LIN {X 0,Y 573.521,Z 268.884,A -85,B 0,C 180,E1 -2263.87,E2 -2263.87} C_VEL
LIN {X 0,Y 573.772,Z 242.194,A -85,B 0,C 180,E1 -2266.729,E2 -2266.729} C_VEL
LIN {X 0,Y 574.13,Z 213.422,A -85,B 0,C 180,E1 -2269.871,E2 -2269.871} C_VEL
LIN {X 0,Y 574.348,Z 185.649,A -85,B 0,C 180,E1 -2272.862,E2 -2272.862} C_VEL
LIN {X 0,Y 574.24,Z 177.963,A -85,B 0,C 180,E1 -2273.69,E2 -2273.69} C_VEL
LIN {X 0,Y 573.256,Z 173.17,A -85,B 0,C 180,E1 -2274.273,E2 -2274.273} C_VEL
LIN {X 0,Y 573.202,Z 173.086,A -85,B 0,C 180,E1 -2276.979,E2 -2276.979} C_VEL
LIN {X 0,Y 573.224,Z 173.084,A -85,B 0,C 180,E1 -2279.484,E2 -2279.484} C_VEL
LIN {X 0,Y 573.24,Z 173.075,A -85,B 0,C 180,E1 -2282.226,E2 -2282.226} C_VEL
LIN {X 0,Y 573.231,Z 173.08,A -85,B 0,C 180,E1 -2284.77,E2 -2284.77} C_VEL
LIN {X 0,Y 573.23,Z 173.077,A -85,B 0,C 180,E1 -2287.808,E2 -2287.808} C_VEL
LIN {X 0,Y 573.248,Z 173.076,A -85,B 0,C 180,E1 -2290.525,E2 -2290.525} C_VEL
LIN {X 0,Y 573.237,Z 173.076,A -85,B 0,C 180,E1 -2293.668,E2 -2293.668} C_VEL
LIN {X 0,Y 573.211,Z 173.083,A -85,B 0,C 180,E1 -2296.638,E2 -2296.638} C_VEL
LIN {X 0,Y 573.247,Z 173.075,A -85,B 0,C 180,E1 -2299.475,E2 -2299.475} C_VEL
LIN {X 0,Y 573.233,Z 173.076,A -85,B 0,C 180,E1 -2302.192,E2 -2302.192} C_VEL
LIN {X 0,Y 573.235,Z 173.079,A -85,B 0,C 180,E1 -2305.229,E2 -2305.229} C_VEL
LIN {X 0,Y 573.238,Z 173.076,A -85,B 0,C 180,E1 -2308.184,E2 -2308.184} C_VEL
LIN {X 0,Y 573.258,Z 173.081,A -85,B 0,C 180,E1 -2310.633,E2 -2310.633} C_VEL
LIN {X 0,Y 573.235,Z 173.075,A -85,B 0,C 180,E1 -2313.508,E2 -2313.508} C_VEL
LIN {X 0,Y 573.227,Z 173.079,A -85,B 0,C 180,E1 -2316.134,E2 -2316.134} C_VEL
LIN {X 0,Y 573.25,Z 173.075,A -85,B 0,C 180,E1 -2319.173,E2 -2319.173} C_VEL
LIN {X 0,Y 573.216,Z 173.078,A -85,B 0,C 180,E1 -2321.411,E2 -2321.411} C_VEL
LIN {X 0,Y 573.244,Z 173.074,A -85,B 0,C 180,E1 -2323.621,E2 -2323.621} C_VEL
LIN {X 0,Y 573.266,Z 173.073,A -85,B 0,C 180,E1 -2325.807,E2 -2325.807} C_VEL
LIN {X 0,Y 573.264,Z 173.077,A -85,B 0,C 180,E1 -2328.745,E2 -2328.745} C_VEL
LIN {X 0,Y 573.253,Z 173.073,A -85,B 0,C 180,E1 -2331.54,E2 -2331.54} C_VEL
LIN {X 0,Y 573.286,Z 173.078,A -85,B 0,C 180,E1 -2334.371,E2 -2334.371} C_VEL
LIN {X 0,Y 573.304,Z 173.072,A -85,B 0,C 180,E1 -2337.892,E2 -2337.892} C_VEL
LIN {X 0,Y 573.343,Z 173.26,A -85,B 0,C 180,E1 -2340.109,E2 -2340.109} C_VEL
LIN {X 0,Y 573.407,Z 187.13,A -85,B 0,C 180,E1 -2342.458,E2 -2342.458} C_VEL
LIN {X 0,Y 573.297,Z 202.339,A -85,B 0,C 180,E1 -2345.275,E2 -2345.275} C_VEL
LIN {X 0,Y 573.189,Z 217.748,A -85,B 0,C 180,E1 -2348.106,E2 -2348.106} C_VEL
LIN {X 0,Y 573.156,Z 223.495,A -85,B 0,C 180,E1 -2349.128,E2 -2349.128} C_VEL
LIN {X 0,Y 573.287,Z 224.818,A -85,B 0,C 180,E1 -2349.192,E2 -2349.192} C_VEL
LIN {X 0,Y 573.63,Z 230.578,A -85,B 0,C 180,E1 -2349.275,E2 -2349.275} C_VEL
LIN {X 0,Y 573.567,Z 299.116,A -85,B 0,C 180,E1 -2350.145,E2 -2350.145} C_VEL
LIN {X 0,Y 573.504,Z 308.495,A -85,B 0,C 180,E1 -2350.346,E2 -2350.346} C_VEL
LIN {X 0,Y 573.472,Z 317.469,A -85,B 0,C 180,E1 -2350.632,E2 -2350.632} C_VEL
LIN {X 0,Y 573.416,Z 327.573,A -85,B 0,C 180,E1 -2351.07,E2 -2351.07} C_VEL
LIN {X 0,Y 573.32,Z 337.992,A -85,B 0,C 180,E1 -2351.669,E2 -2351.669} C_VEL
LIN {X 0,Y 573.19,Z 347.471,A -85,B 0,C 180,E1 -2352.39,E2 -2352.39} C_VEL
LIN {X 0,Y 573.167,Z 353.388,A -85,B 0,C 180,E1 -2352.934,E2 -2352.934} C_VEL
LIN {X 0,Y 572.469,Z 357.587,A -85,B 0,C 180,E1 -2353.364,E2 -2353.364} C_VEL
LIN {X 0,Y 569.555,Z 363.708,A -85,B 0,C 180,E1 -2354.095,E2 -2354.095} C_VEL
LIN {X 0,Y 566.642,Z 369.015,A -85,B 0,C 180,E1 -2354.883,E2 -2354.883} C_VEL
LIN {X 0,Y 565.93,Z 371.801,A -85,B 0,C 180,E1 -2355.396,E2 -2355.396} C_VEL
LIN {X 0,Y 565.894,Z 376.999,A -85,B 0,C 180,E1 -2356.597,E2 -2356.597} C_VEL
LIN {X 0,Y 565.863,Z 379.373,A -85,B 0,C 180,E1 -2357.342,E2 -2357.342} C_VEL
LIN {X 0,Y 565.836,Z 381.091,A -85,B 0,C 180,E1 -2358.09,E2 -2358.09} C_VEL
LIN {X 0,Y 565.87,Z 382.685,A -85,B 0,C 180,E1 -2359.282,E2 -2359.282} C_VEL
LIN {X 0,Y 565.832,Z 382.89,A -85,B 0,C 180,E1 -2360.351,E2 -2360.351} C_VEL
LIN {X 0,Y 565.862,Z 382.12,A -85,B 0,C 180,E1 -2361.331,E2 -2361.331} C_VEL
LIN {X 0,Y 565.835,Z 381.35,A -85,B 0,C 180,E1 -2361.877,E2 -2361.877} C_VEL
LIN {X 0,Y 565.872,Z 379.63,A -85,B 0,C 180,E1 -2362.644,E2 -2362.644} C_VEL
LIN {X 0,Y 565.916,Z 375.822,A -85,B 0,C 180,E1 -2363.804,E2 -2363.804} C_VEL
LIN {X 0,Y 565.944,Z 371.347,A -85,B 0,C 180,E1 -2364.778,E2 -2364.778} C_VEL
LIN {X 0,Y 565.966,Z 366.81,A -85,B 0,C 180,E1 -2365.563,E2 -2365.563} C_VEL
LIN {X 0,Y 566.035,Z 361.227,A -85,B 0,C 180,E1 -2366.351,E2 -2366.351} C_VEL
LIN {X 0,Y 566.065,Z 356.174,A -85,B 0,C 180,E1 -2366.953,E2 -2366.953} C_VEL
LIN {X 0,Y 566.142,Z 349.213,A -85,B 0,C 180,E1 -2367.643,E2 -2367.643} C_VEL
LIN {X 0,Y 566.219,Z 342.41,A -85,B 0,C 180,E1 -2368.205,E2 -2368.205} C_VEL
LIN {X 0,Y 566.291,Z 334.823,A -85,B 0,C 180,E1 -2368.724,E2 -2368.724} C_VEL
LIN {X 0,Y 566.376,Z 326.258,A -85,B 0,C 180,E1 -2369.197,E2 -2369.197} C_VEL
LIN {X 0,Y 566.464,Z 316.793,A -85,B 0,C 180,E1 -2369.601,E2 -2369.601} C_VEL
LIN {X 0,Y 566.533,Z 307.068,A -85,B 0,C 180,E1 -2369.903,E2 -2369.903} C_VEL
LIN {X 0,Y 566.574,Z 295.422,A -85,B 0,C 180,E1 -2370.131,E2 -2370.131} C_VEL
LIN {X 0,Y 566.574,Z 227.134,A -85,B 0,C 180,E1 -2370.994,E2 -2370.994} C_VEL
LIN {X 0,Y 566.123,Z 223.733,A -85,B 0,C 180,E1 -2371.08,E2 -2371.08} C_VEL
LIN {X 0,Y 566.129,Z 219.328,A -85,B 0,C 180,E1 -2371.843,E2 -2371.843} C_VEL
LIN {X 0,Y 566.266,Z 203.344,A -85,B 0,C 180,E1 -2374.813,E2 -2374.813} C_VEL
LIN {X 0,Y 566.371,Z 187.85,A -85,B 0,C 180,E1 -2377.671,E2 -2377.671} C_VEL
LIN {X 0,Y 566.432,Z 175.809,A -85,B 0,C 180,E1 -2379.916,E2 -2379.916} C_VEL
LIN {X 0,Y 566.271,Z 173.97,A -85,B 0,C 180,E1 -2380.331,E2 -2380.331} C_VEL
LIN {X 0,Y 566.198,Z 173.953,A -85,B 0,C 180,E1 -2383.054,E2 -2383.054} C_VEL
LIN {X 0,Y 566.197,Z 173.958,A -85,B 0,C 180,E1 -2386.048,E2 -2386.048} C_VEL
LIN {X 0,Y 566.177,Z 173.954,A -85,B 0,C 180,E1 -2388.861,E2 -2388.861} C_VEL
LIN {X 0,Y 566.184,Z 173.962,A -85,B 0,C 180,E1 -2391.637,E2 -2391.637} C_VEL
LIN {X 0,Y 566.195,Z 173.953,A -85,B 0,C 180,E1 -2394.31,E2 -2394.31} C_VEL
LIN {X 0,Y 566.219,Z 173.949,A -85,B 0,C 180,E1 -2396.898,E2 -2396.898} C_VEL
LIN {X 0,Y 566.179,Z 173.961,A -85,B 0,C 180,E1 -2399.407,E2 -2399.407} C_VEL
LIN {X 0,Y 566.21,Z 173.954,A -85,B 0,C 180,E1 -2401.857,E2 -2401.857} C_VEL
LIN {X 0,Y 566.224,Z 173.948,A -85,B 0,C 180,E1 -2404.251,E2 -2404.251} C_VEL
LIN {X 0,Y 566.172,Z 173.955,A -85,B 0,C 180,E1 -2406.718,E2 -2406.718} C_VEL
LIN {X 0,Y 566.207,Z 173.956,A -85,B 0,C 180,E1 -2409.662,E2 -2409.662} C_VEL
LIN {X 0,Y 566.198,Z 173.952,A -85,B 0,C 180,E1 -2412.668,E2 -2412.668} C_VEL
LIN {X 0,Y 566.233,Z 173.952,A -85,B 0,C 180,E1 -2415.626,E2 -2415.626} C_VEL
LIN {X 0,Y 566.233,Z 173.949,A -85,B 0,C 180,E1 -2418.675,E2 -2418.675} C_VEL
LIN {X 0,Y 566.231,Z 173.953,A -85,B 0,C 180,E1 -2421.434,E2 -2421.434} C_VEL
LIN {X 0,Y 566.264,Z 173.943,A -85,B 0,C 180,E1 -2424.301,E2 -2424.301} C_VEL
LIN {X 0,Y 566.284,Z 173.941,A -85,B 0,C 180,E1 -2427.866,E2 -2427.866} C_VEL
LIN {X 0,Y 566.298,Z 173.943,A -85,B 0,C 180,E1 -2430.711,E2 -2430.711} C_VEL
LIN {X 0,Y 566.268,Z 173.949,A -85,B 0,C 180,E1 -2432.845,E2 -2432.845} C_VEL
LIN {X 0,Y 566.263,Z 173.944,A -85,B 0,C 180,E1 -2435.698,E2 -2435.698} C_VEL
LIN {X 0,Y 566.225,Z 173.952,A -85,B 0,C 180,E1 -2438.565,E2 -2438.565} C_VEL
LIN {X 0,Y 566.239,Z 173.948,A -85,B 0,C 180,E1 -2441.454,E2 -2441.454} C_VEL
LIN {X 0,Y 566.231,Z 173.951,A -85,B 0,C 180,E1 -2444.506,E2 -2444.506} C_VEL
LIN {X 0,Y 566.196,Z 173.954,A -85,B 0,C 180,E1 -2447.331,E2 -2447.331} C_VEL
LIN {X 0,Y 566.209,Z 173.953,A -85,B 0,C 180,E1 -2450.337,E2 -2450.337} C_VEL
LIN {X 0,Y 566.185,Z 173.954,A -85,B 0,C 180,E1 -2453.403,E2 -2453.403} C_VEL
LIN {X 0,Y 566.221,Z 173.948,A -85,B 0,C 180,E1 -2455.748,E2 -2455.748} C_VEL
LIN {X 0,Y 566.202,Z 173.954,A -85,B 0,C 180,E1 -2458.203,E2 -2458.203} C_VEL
LIN {X 0,Y 566.193,Z 173.955,A -85,B 0,C 180,E1 -2461.077,E2 -2461.077} C_VEL
LIN {X 0,Y 566.216,Z 173.951,A -85,B 0,C 180,E1 -2463.955,E2 -2463.955} C_VEL
LIN {X 0,Y 566.21,Z 173.959,A -85,B 0,C 180,E1 -2466.568,E2 -2466.568} C_VEL
LIN {X 0,Y 566.206,Z 173.951,A -85,B 0,C 180,E1 -2469.685,E2 -2469.685} C_VEL
LIN {X 0,Y 566.207,Z 173.955,A -85,B 0,C 180,E1 -2472.087,E2 -2472.087} C_VEL
LIN {X 0,Y 566.165,Z 173.956,A -85,B 0,C 180,E1 -2475.035,E2 -2475.035} C_VEL
LIN {X 0,Y 566.21,Z 173.956,A -85,B 0,C 180,E1 -2478.135,E2 -2478.135} C_VEL
LIN {X 0,Y 566.215,Z 173.952,A -85,B 0,C 180,E1 -2480.727,E2 -2480.727} C_VEL
LIN {X 0,Y 566.21,Z 173.953,A -85,B 0,C 180,E1 -2483.783,E2 -2483.783} C_VEL
LIN {X 0,Y 566.221,Z 173.957,A -85,B 0,C 180,E1 -2486.263,E2 -2486.263} C_VEL
LIN {X 0,Y 566.194,Z 173.952,A -85,B 0,C 180,E1 -2488.921,E2 -2488.921} C_VEL
LIN {X 0,Y 566.189,Z 173.952,A -85,B 0,C 180,E1 -2491.047,E2 -2491.047} C_VEL
LIN {X 0,Y 566.208,Z 173.951,A -85,B 0,C 180,E1 -2493.459,E2 -2493.459} C_VEL
LIN {X 0,Y 566.191,Z 173.958,A -85,B 0,C 180,E1 -2495.819,E2 -2495.819} C_VEL
LIN {X 0,Y 566.208,Z 173.95,A -85,B 0,C 180,E1 -2498.903,E2 -2498.903} C_VEL
LIN {X 0,Y 566.205,Z 173.951,A -85,B 0,C 180,E1 -2501.173,E2 -2501.173} C_VEL
LIN {X 0,Y 566.212,Z 173.952,A -85,B 0,C 180,E1 -2503.413,E2 -2503.413} C_VEL
LIN {X 0,Y 566.19,Z 173.955,A -85,B 0,C 180,E1 -2506.359,E2 -2506.359} C_VEL
LIN {X 0,Y 566.267,Z 173.943,A -85,B 0,C 180,E1 -2508.654,E2 -2508.654} C_VEL
LIN {X 0,Y 566.225,Z 173.952,A -85,B 0,C 180,E1 -2511.435,E2 -2511.435} C_VEL
LIN {X 0,Y 566.248,Z 173.947,A -85,B 0,C 180,E1 -2514.302,E2 -2514.302} C_VEL
LIN {X 0,Y 566.269,Z 173.95,A -85,B 0,C 180,E1 -2517.867,E2 -2517.867} C_VEL
LIN {X 0,Y 566.293,Z 173.939,A -85,B 0,C 180,E1 -2520.711,E2 -2520.711} C_VEL
LIN {X 0,Y 566.264,Z 173.943,A -85,B 0,C 180,E1 -2522.846,E2 -2522.846} C_VEL
LIN {X 0,Y 566.251,Z 173.953,A -85,B 0,C 180,E1 -2525.699,E2 -2525.699} C_VEL
LIN {X 0,Y 566.198,Z 173.951,A -85,B 0,C 180,E1 -2528.566,E2 -2528.566} C_VEL
LIN {X 0,Y 566.234,Z 173.956,A -85,B 0,C 180,E1 -2531.455,E2 -2531.455} C_VEL
LIN {X 0,Y 566.222,Z 173.948,A -85,B 0,C 180,E1 -2534.505,E2 -2534.505} C_VEL
LIN {X 0,Y 566.191,Z 173.961,A -85,B 0,C 180,E1 -2537.332,E2 -2537.332} C_VEL
LIN {X 0,Y 566.199,Z 173.951,A -85,B 0,C 180,E1 -2540.338,E2 -2540.338} C_VEL
LIN {X 0,Y 566.165,Z 173.965,A -85,B 0,C 180,E1 -2543.282,E2 -2543.282} C_VEL
LIN {X 0,Y 566.202,Z 173.954,A -85,B 0,C 180,E1 -2545.75,E2 -2545.75} C_VEL
LIN {X 0,Y 566.196,Z 173.951,A -85,B 0,C 180,E1 -2548.203,E2 -2548.203} C_VEL
LIN {X 0,Y 566.187,Z 173.961,A -85,B 0,C 180,E1 -2551.077,E2 -2551.077} C_VEL
LIN {X 0,Y 566.191,Z 173.954,A -85,B 0,C 180,E1 -2553.733,E2 -2553.733} C_VEL
LIN {X 0,Y 566.194,Z 173.954,A -85,B 0,C 180,E1 -2556.571,E2 -2556.571} C_VEL
LIN {X 0,Y 566.208,Z 173.951,A -85,B 0,C 180,E1 -2559.686,E2 -2559.686} C_VEL
LIN {X 0,Y 566.194,Z 173.96,A -85,B 0,C 180,E1 -2562.918,E2 -2562.918} C_VEL
LIN {X 0,Y 566.189,Z 173.952,A -85,B 0,C 180,E1 -2566.05,E2 -2566.05} C_VEL
LIN {X 0,Y 566.199,Z 173.956,A -85,B 0,C 180,E1 -2569.216,E2 -2569.216} C_VEL
LIN {X 0,Y 566.18,Z 173.954,A -85,B 0,C 180,E1 -2571.637,E2 -2571.637} C_VEL
LIN {X 0,Y 566.147,Z 173.96,A -85,B 0,C 180,E1 -2574.308,E2 -2574.308} C_VEL
LIN {X 0,Y 566.207,Z 173.959,A -85,B 0,C 180,E1 -2576.898,E2 -2576.898} C_VEL
LIN {X 0,Y 566.167,Z 173.958,A -85,B 0,C 180,E1 -2579.407,E2 -2579.407} C_VEL
LIN {X 0,Y 566.187,Z 173.955,A -85,B 0,C 180,E1 -2581.857,E2 -2581.857} C_VEL
LIN {X 0,Y 566.194,Z 173.959,A -85,B 0,C 180,E1 -2584.251,E2 -2584.251} C_VEL
LIN {X 0,Y 566.221,Z 174.083,A -85,B 0,C 180,E1 -2585.455,E2 -2585.455} C_VEL
LIN {X 0,Y 567.5,Z 179.942,A -85,B 0,C 180,E1 -2586.196,E2 -2586.196} C_VEL
LIN {X 0,Y 567.326,Z 199.749,A -85,B 0,C 180,E1 -2588.415,E2 -2588.415} C_VEL
LIN {X 0,Y 567.012,Z 225.162,A -85,B 0,C 180,E1 -2591.201,E2 -2591.201} C_VEL
LIN {X 0,Y 566.776,Z 248.942,A -85,B 0,C 180,E1 -2593.8,E2 -2593.8} C_VEL
LIN {X 0,Y 566.566,Z 268.903,A -85,B 0,C 180,E1 -2595.957,E2 -2595.957} C_VEL
LIN {X 0,Y 567.141,Z 274.771,A -85,B 0,C 180,E1 -2596.063,E2 -2596.063} C_VEL
LIN {X 0,Y 566.98,Z 378.978,A -85,B 0,C 180,E1 -2597.404,E2 -2597.404} C_VEL
LIN {X 0,Y 566.87,Z 392.239,A -85,B 0,C 180,E1 -2597.72,E2 -2597.72} C_VEL
LIN {X 0,Y 566.731,Z 405.171,A -85,B 0,C 180,E1 -2598.18,E2 -2598.18} C_VEL
LIN {X 0,Y 566.611,Z 417.257,A -85,B 0,C 180,E1 -2598.771,E2 -2598.771} C_VEL
LIN {X 0,Y 566.422,Z 429.493,A -85,B 0,C 180,E1 -2599.546,E2 -2599.546} C_VEL
LIN {X 0,Y 566.299,Z 439.653,A -85,B 0,C 180,E1 -2600.356,E2 -2600.356} C_VEL
LIN {X 0,Y 566.166,Z 448.791,A -85,B 0,C 180,E1 -2601.254,E2 -2601.254} C_VEL
LIN {X 0,Y 566.08,Z 457.693,A -85,B 0,C 180,E1 -2602.331,E2 -2602.331} C_VEL
LIN {X 0,Y 565.967,Z 464.959,A -85,B 0,C 180,E1 -2603.423,E2 -2603.423} C_VEL
LIN {X 0,Y 566.004,Z 469.682,A -85,B 0,C 180,E1 -2604.3,E2 -2604.3} C_VEL
LIN {X 0,Y 565.933,Z 474.375,A -85,B 0,C 180,E1 -2605.371,E2 -2605.371} C_VEL
LIN {X 0,Y 565.927,Z 477.959,A -85,B 0,C 180,E1 -2606.441,E2 -2606.441} C_VEL
LIN {X 0,Y 565.878,Z 479.809,A -85,B 0,C 180,E1 -2607.153,E2 -2607.153} C_VEL
LIN {X 0,Y 565.846,Z 482.185,A -85,B 0,C 180,E1 -2608.577,E2 -2608.577} C_VEL
LIN {X 0,Y 565.839,Z 483,A -85,B 0,C 180,E1 -2610,E2 -2610} C_VEL
LIN {X 0,Y 565.846,Z 482.185,A -85,B 0,C 180,E1 -2611.424,E2 -2611.424} C_VEL
LIN {X 0,Y 565.878,Z 479.809,A -85,B 0,C 180,E1 -2612.848,E2 -2612.848} C_VEL
LIN {X 0,Y 565.926,Z 476.894,A -85,B 0,C 180,E1 -2613.917,E2 -2613.917} C_VEL
LIN {X 0,Y 565.878,Z 472.947,A -85,B 0,C 180,E1 -2614.988,E2 -2614.988} C_VEL
LIN {X 0,Y 566.002,Z 467.865,A -85,B 0,C 180,E1 -2616.059,E2 -2616.059} C_VEL
LIN {X 0,Y 566.041,Z 461.465,A -85,B 0,C 180,E1 -2617.133,E2 -2617.133} C_VEL
LIN {X 0,Y 566.134,Z 453.474,A -85,B 0,C 180,E1 -2618.208,E2 -2618.208} C_VEL
LIN {X 0,Y 566.229,Z 445.33,A -85,B 0,C 180,E1 -2619.106,E2 -2619.106} C_VEL
LIN {X 0,Y 566.351,Z 435.394,A -85,B 0,C 180,E1 -2620.005,E2 -2620.005} C_VEL
LIN {X 0,Y 566.529,Z 424.285,A -85,B 0,C 180,E1 -2620.808,E2 -2620.808} C_VEL
LIN {X 0,Y 566.614,Z 413.166,A -85,B 0,C 180,E1 -2621.447,E2 -2621.447} C_VEL
LIN {X 0,Y 566.75,Z 400.97,A -85,B 0,C 180,E1 -2621.988,E2 -2621.988} C_VEL
LIN {X 0,Y 566.889,Z 388.159,A -85,B 0,C 180,E1 -2622.394,E2 -2622.394} C_VEL
LIN {X 0,Y 566.968,Z 374.575,A -85,B 0,C 180,E1 -2622.665,E2 -2622.665} C_VEL
LIN {X 0,Y 567.07,Z 272.9,A -85,B 0,C 180,E1 -2623.963,E2 -2623.963} C_VEL
LIN {X 0,Y 566.566,Z 268.885,A -85,B 0,C 180,E1 -2624.044,E2 -2624.044} C_VEL
LIN {X 0,Y 566.852,Z 241.138,A -85,B 0,C 180,E1 -2627.056,E2 -2627.056} C_VEL
LIN {X 0,Y 567.136,Z 214.637,A -85,B 0,C 180,E1 -2629.924,E2 -2629.924} C_VEL
LIN {X 0,Y 567.397,Z 186.667,A -85,B 0,C 180,E1 -2632.965,E2 -2632.965} C_VEL
LIN {X 0,Y 567.228,Z 178.993,A -85,B 0,C 180,E1 -2633.804,E2 -2633.804} C_VEL
LIN {X 0,Y 566.23,Z 174.085,A -85,B 0,C 180,E1 -2634.399,E2 -2634.399} C_VEL
LIN {X 0,Y 566.174,Z 173.964,A -85,B 0,C 180,E1 -2637.341,E2 -2637.341} C_VEL
LIN {X 0,Y 566.172,Z 173.959,A -85,B 0,C 180,E1 -2639.771,E2 -2639.771} C_VEL
LIN {X 0,Y 566.195,Z 173.953,A -85,B 0,C 180,E1 -2642.428,E2 -2642.428} C_VEL
LIN {X 0,Y 566.178,Z 173.962,A -85,B 0,C 180,E1 -2644.989,E2 -2644.989} C_VEL
LIN {X 0,Y 566.194,Z 173.957,A -85,B 0,C 180,E1 -2647.461,E2 -2647.461} C_VEL
LIN {X 0,Y 566.208,Z 173.951,A -85,B 0,C 180,E1 -2650.199,E2 -2650.199} C_VEL
LIN {X 0,Y 566.195,Z 173.962,A -85,B 0,C 180,E1 -2653.055,E2 -2653.055} C_VEL
LIN {X 0,Y 566.161,Z 173.956,A -85,B 0,C 180,E1 -2656.053,E2 -2656.053} C_VEL
LIN {X 0,Y 566.17,Z 173.964,A -85,B 0,C 180,E1 -2658.86,E2 -2658.86} C_VEL
LIN {X 0,Y 566.208,Z 173.952,A -85,B 0,C 180,E1 -2661.442,E2 -2661.442} C_VEL
LIN {X 0,Y 566.163,Z 173.958,A -85,B 0,C 180,E1 -2664.308,E2 -2664.308} C_VEL
LIN {X 0,Y 566.202,Z 173.96,A -85,B 0,C 180,E1 -2666.896,E2 -2666.896} C_VEL
LIN {X 0,Y 566.173,Z 173.956,A -85,B 0,C 180,E1 -2669.406,E2 -2669.406} C_VEL
LIN {X 0,Y 566.195,Z 173.952,A -85,B 0,C 180,E1 -2671.856,E2 -2671.856} C_VEL
LIN {X 0,Y 566.208,Z 173.954,A -85,B 0,C 180,E1 -2674.25,E2 -2674.25} C_VEL
LIN {X 0,Y 566.172,Z 173.963,A -85,B 0,C 180,E1 -2676.718,E2 -2676.718} C_VEL
LIN {X 0,Y 566.206,Z 173.951,A -85,B 0,C 180,E1 -2679.662,E2 -2679.662} C_VEL
LIN {X 0,Y 566.199,Z 173.96,A -85,B 0,C 180,E1 -2682.668,E2 -2682.668} C_VEL
LIN {X 0,Y 566.229,Z 173.948,A -85,B 0,C 180,E1 -2685.626,E2 -2685.626} C_VEL
LIN {X 0,Y 566.236,Z 173.953,A -85,B 0,C 180,E1 -2688.675,E2 -2688.675} C_VEL
LIN {X 0,Y 566.204,Z 173.951,A -85,B 0,C 180,E1 -2691.434,E2 -2691.434} C_VEL
LIN {X 0,Y 566.253,Z 173.954,A -85,B 0,C 180,E1 -2694.301,E2 -2694.301} C_VEL
LIN {X 0,Y 566.275,Z 173.947,A -85,B 0,C 180,E1 -2697.866,E2 -2697.866} C_VEL
LIN {X 0,Y 566.295,Z 174.105,A -85,B 0,C 180,E1 -2700.222,E2 -2700.222} C_VEL
LIN {X 0,Y 566.323,Z 185.594,A -85,B 0,C 180,E1 -2702.133,E2 -2702.133} C_VEL
LIN {X 0,Y 566.265,Z 199.749,A -85,B 0,C 180,E1 -2704.627,E2 -2704.627} C_VEL
LIN {X 0,Y 566.13,Z 215.239,A -85,B 0,C 180,E1 -2707.489,E2 -2707.489} C_VEL
LIN {X 0,Y 566.096,Z 223.554,A -85,B 0,C 180,E1 -2708.995,E2 -2708.995} C_VEL
LIN {X 0,Y 566.255,Z 225.049,A -85,B 0,C 180,E1 -2709.06,E2 -2709.06} C_VEL
LIN {X 0,Y 566.673,Z 230.673,A -85,B 0,C 180,E1 -2709.143,E2 -2709.143} C_VEL
LIN {X 0,Y 566.592,Z 299.184,A -85,B 0,C 180,E1 -2710.023,E2 -2710.023} C_VEL
LIN {X 0,Y 566.503,Z 308.568,A -85,B 0,C 180,E1 -2710.227,E2 -2710.227} C_VEL
LIN {X 0,Y 566.459,Z 318.268,A -85,B 0,C 180,E1 -2710.544,E2 -2710.544} C_VEL
LIN {X 0,Y 566.398,Z 328.843,A -85,B 0,C 180,E1 -2711.019,E2 -2711.019} C_VEL
LIN {X 0,Y 566.257,Z 338.974,A -85,B 0,C 180,E1 -2711.635,E2 -2711.635} C_VEL
LIN {X 0,Y 566.177,Z 347.221,A -85,B 0,C 180,E1 -2712.273,E2 -2712.273} C_VEL
LIN {X 0,Y 566.112,Z 354.026,A -85,B 0,C 180,E1 -2712.912,E2 -2712.912} C_VEL
LIN {X 0,Y 566.056,Z 360.479,A -85,B 0,C 180,E1 -2713.644,E2 -2713.644} C_VEL
LIN {X 0,Y 566.004,Z 366.081,A -85,B 0,C 180,E1 -2714.416,E2 -2714.416} C_VEL
LIN {X 0,Y 565.965,Z 370.295,A -85,B 0,C 180,E1 -2715.116,E2 -2715.116} C_VEL
LIN {X 0,Y 565.93,Z 371.801,A -85,B 0,C 180,E1 -2715.396,E2 -2715.396} C_VEL
LIN {X 0,Y 565.218,Z 374.462,A -85,B 0,C 180,E1 -2715.928,E2 -2715.928} C_VEL
LIN {X 0,Y 562.298,Z 378.055,A -85,B 0,C 180,E1 -2716.823,E2 -2716.823} C_VEL
LIN {X 0,Y 559.4,Z 380.595,A -85,B 0,C 180,E1 -2717.762,E2 -2717.762} C_VEL
LIN {X 0,Y 558.73,Z 381.603,A -85,B 0,C 180,E1 -2718.358,E2 -2718.358} C_VEL
LIN {X 0,Y 558.767,Z 382.733,A -85,B 0,C 180,E1 -2719.382,E2 -2719.382} C_VEL
LIN {X 0,Y 558.742,Z 382.772,A -85,B 0,C 180,E1 -2720.621,E2 -2720.621} C_VEL
LIN {X 0,Y 558.768,Z 381.983,A -85,B 0,C 180,E1 -2721.449,E2 -2721.449} C_VEL
LIN {X 0,Y 558.753,Z 380.771,A -85,B 0,C 180,E1 -2722.169,E2 -2722.169} C_VEL
LIN {X 0,Y 558.802,Z 377.599,A -85,B 0,C 180,E1 -2723.348,E2 -2723.348} C_VEL
LIN {X 0,Y 558.815,Z 374.671,A -85,B 0,C 180,E1 -2724.125,E2 -2724.125} C_VEL
LIN {X 0,Y 558.852,Z 371.446,A -85,B 0,C 180,E1 -2724.82,E2 -2724.82} C_VEL
LIN {X 0,Y 558.904,Z 366.312,A -85,B 0,C 180,E1 -2725.71,E2 -2725.71} C_VEL
LIN {X 0,Y 558.981,Z 360.62,A -85,B 0,C 180,E1 -2726.508,E2 -2726.508} C_VEL
LIN {X 0,Y 559.015,Z 355.499,A -85,B 0,C 180,E1 -2727.112,E2 -2727.112} C_VEL
LIN {X 0,Y 559.099,Z 348.338,A -85,B 0,C 180,E1 -2727.817,E2 -2727.817} C_VEL
LIN {X 0,Y 559.169,Z 341.423,A -85,B 0,C 180,E1 -2728.381,E2 -2728.381} C_VEL
LIN {X 0,Y 559.309,Z 333.196,A -85,B 0,C 180,E1 -2728.932,E2 -2728.932} C_VEL
LIN {X 0,Y 559.408,Z 323.85,A -85,B 0,C 180,E1 -2729.429,E2 -2729.429} C_VEL
LIN {X 0,Y 559.544,Z 312.135,A -85,B 0,C 180,E1 -2729.888,E2 -2729.888} C_VEL
LIN {X 0,Y 559.59,Z 301.336,A -85,B 0,C 180,E1 -2730.156,E2 -2730.156} C_VEL
LIN {X 0,Y 559.599,Z 274.915,A -85,B 0,C 180,E1 -2730.521,E2 -2730.521} C_VEL
LIN {X 0,Y 559.625,Z 227.896,A -85,B 0,C 180,E1 -2731.122,E2 -2731.122} C_VEL
LIN {X 0,Y 559.088,Z 223.909,A -85,B 0,C 180,E1 -2731.21,E2 -2731.21} C_VEL
LIN {X 0,Y 559.062,Z 221.829,A -85,B 0,C 180,E1 -2731.53,E2 -2731.53} C_VEL
LIN {X 0,Y 559.225,Z 206.44,A -85,B 0,C 180,E1 -2734.439,E2 -2734.439} C_VEL
LIN {X 0,Y 559.314,Z 190.38,A -85,B 0,C 180,E1 -2737.382,E2 -2737.382} C_VEL
LIN {X 0,Y 559.406,Z 176.654,A -85,B 0,C 180,E1 -2739.972,E2 -2739.972} C_VEL
LIN {X 0,Y 559.225,Z 174.852,A -85,B 0,C 180,E1 -2740.376,E2 -2740.376} C_VEL
LIN {X 0,Y 559.143,Z 174.833,A -85,B 0,C 180,E1 -2743.196,E2 -2743.196} C_VEL
LIN {X 0,Y 559.14,Z 174.834,A -85,B 0,C 180,E1 -2746.266,E2 -2746.266} C_VEL
LIN {X 0,Y 559.164,Z 174.828,A -85,B 0,C 180,E1 -2748.948,E2 -2748.948} C_VEL
LIN {X 0,Y 559.172,Z 174.829,A -85,B 0,C 180,E1 -2751.191,E2 -2751.191} C_VEL
LIN {X 0,Y 559.159,Z 174.835,A -85,B 0,C 180,E1 -2753.791,E2 -2753.791} C_VEL
LIN {X 0,Y 559.161,Z 174.828,A -85,B 0,C 180,E1 -2756.425,E2 -2756.425} C_VEL
LIN {X 0,Y 559.153,Z 174.831,A -85,B 0,C 180,E1 -2758.98,E2 -2758.98} C_VEL
LIN {X 0,Y 559.167,Z 174.836,A -85,B 0,C 180,E1 -2761.618,E2 -2761.618} C_VEL
LIN {X 0,Y 559.197,Z 174.827,A -85,B 0,C 180,E1 -2763.903,E2 -2763.903} C_VEL
LIN {X 0,Y 559.141,Z 174.83,A -85,B 0,C 180,E1 -2766.57,E2 -2766.57} C_VEL
LIN {X 0,Y 559.176,Z 174.836,A -85,B 0,C 180,E1 -2769.395,E2 -2769.395} C_VEL
LIN {X 0,Y 559.143,Z 174.835,A -85,B 0,C 180,E1 -2771.685,E2 -2771.685} C_VEL
LIN {X 0,Y 559.165,Z 174.829,A -85,B 0,C 180,E1 -2773.947,E2 -2773.947} C_VEL
LIN {X 0,Y 559.17,Z 174.827,A -85,B 0,C 180,E1 -2776.184,E2 -2776.184} C_VEL
LIN {X 0,Y 559.195,Z 174.832,A -85,B 0,C 180,E1 -2779.133,E2 -2779.133} C_VEL
LIN {X 0,Y 559.204,Z 174.823,A -85,B 0,C 180,E1 -2782.053,E2 -2782.053} C_VEL
LIN {X 0,Y 559.253,Z 174.823,A -85,B 0,C 180,E1 -2784.953,E2 -2784.953} C_VEL
LIN {X 0,Y 559.255,Z 174.817,A -85,B 0,C 180,E1 -2787.839,E2 -2787.839} C_VEL
LIN {X 0,Y 559.269,Z 174.819,A -85,B 0,C 180,E1 -2790.72,E2 -2790.72} C_VEL
LIN {X 0,Y 559.235,Z 174.826,A -85,B 0,C 180,E1 -2792.881,E2 -2792.881} C_VEL
LIN {X 0,Y 559.231,Z 174.82,A -85,B 0,C 180,E1 -2795.77,E2 -2795.77} C_VEL
LIN {X 0,Y 559.184,Z 174.83,A -85,B 0,C 180,E1 -2798.674,E2 -2798.674} C_VEL
LIN {X 0,Y 559.202,Z 174.824,A -85,B 0,C 180,E1 -2801.6,E2 -2801.6} C_VEL
LIN {X 0,Y 559.196,Z 174.829,A -85,B 0,C 180,E1 -2804.595,E2 -2804.595} C_VEL
LIN {X 0,Y 559.156,Z 174.829,A -85,B 0,C 180,E1 -2807.556,E2 -2807.556} C_VEL
LIN {X 0,Y 559.168,Z 174.827,A -85,B 0,C 180,E1 -2809.837,E2 -2809.837} C_VEL
LIN {X 0,Y 559.137,Z 174.833,A -85,B 0,C 180,E1 -2812.152,E2 -2812.152} C_VEL
LIN {X 0,Y 559.175,Z 174.829,A -85,B 0,C 180,E1 -2815.187,E2 -2815.187} C_VEL
LIN {X 0,Y 559.19,Z 174.824,A -85,B 0,C 180,E1 -2817.711,E2 -2817.711} C_VEL
LIN {X 0,Y 559.157,Z 174.832,A -85,B 0,C 180,E1 -2821.018,E2 -2821.018} C_VEL
LIN {X 0,Y 559.172,Z 174.828,A -85,B 0,C 180,E1 -2823.951,E2 -2823.951} C_VEL
LIN {X 0,Y 559.184,Z 174.834,A -85,B 0,C 180,E1 -2826.451,E2 -2826.451} C_VEL
LIN {X 0,Y 559.171,Z 174.83,A -85,B 0,C 180,E1 -2828.933,E2 -2828.933} C_VEL
LIN {X 0,Y 559.184,Z 174.826,A -85,B 0,C 180,E1 -2831.767,E2 -2831.767} C_VEL
LIN {X 0,Y 559.132,Z 174.836,A -85,B 0,C 180,E1 -2834.739,E2 -2834.739} C_VEL
LIN {X 0,Y 559.153,Z 174.829,A -85,B 0,C 180,E1 -2837.256,E2 -2837.256} C_VEL
LIN {X 0,Y 559.179,Z 174.833,A -85,B 0,C 180,E1 -2840.135,E2 -2840.135} C_VEL
LIN {X 0,Y 559.138,Z 174.832,A -85,B 0,C 180,E1 -2842.892,E2 -2842.892} C_VEL
LIN {X 0,Y 559.153,Z 174.83,A -85,B 0,C 180,E1 -2845.556,E2 -2845.556} C_VEL
LIN {X 0,Y 559.164,Z 174.837,A -85,B 0,C 180,E1 -2848.138,E2 -2848.138} C_VEL
LIN {X 0,Y 559.15,Z 174.832,A -85,B 0,C 180,E1 -2850.647,E2 -2850.647} C_VEL
LIN {X 0,Y 559.162,Z 174.828,A -85,B 0,C 180,E1 -2853.172,E2 -2853.172} C_VEL
LIN {X 0,Y 559.149,Z 174.831,A -85,B 0,C 180,E1 -2855.495,E2 -2855.495} C_VEL
LIN {X 0,Y 559.169,Z 174.828,A -85,B 0,C 180,E1 -2858.624,E2 -2858.624} C_VEL
LIN {X 0,Y 559.163,Z 174.827,A -85,B 0,C 180,E1 -2860.926,E2 -2860.926} C_VEL
LIN {X 0,Y 559.162,Z 174.838,A -85,B 0,C 180,E1 -2863.948,E2 -2863.948} C_VEL
LIN {X 0,Y 559.164,Z 174.833,A -85,B 0,C 180,E1 -2866.184,E2 -2866.184} C_VEL
LIN {X 0,Y 559.202,Z 174.824,A -85,B 0,C 180,E1 -2869.134,E2 -2869.134} C_VEL
LIN {X 0,Y 559.197,Z 174.829,A -85,B 0,C 180,E1 -2872.054,E2 -2872.054} C_VEL
LIN {X 0,Y 559.247,Z 174.818,A -85,B 0,C 180,E1 -2874.954,E2 -2874.954} C_VEL
LIN {X 0,Y 559.241,Z 174.826,A -85,B 0,C 180,E1 -2877.84,E2 -2877.84} C_VEL
LIN {X 0,Y 559.264,Z 174.815,A -85,B 0,C 180,E1 -2880.72,E2 -2880.72} C_VEL
LIN {X 0,Y 559.231,Z 174.82,A -85,B 0,C 180,E1 -2882.882,E2 -2882.882} C_VEL
LIN {X 0,Y 559.219,Z 174.827,A -85,B 0,C 180,E1 -2885.771,E2 -2885.771} C_VEL
LIN {X 0,Y 559.162,Z 174.828,A -85,B 0,C 180,E1 -2888.675,E2 -2888.675} C_VEL
LIN {X 0,Y 559.197,Z 174.831,A -85,B 0,C 180,E1 -2891.601,E2 -2891.601} C_VEL
LIN {X 0,Y 559.192,Z 174.824,A -85,B 0,C 180,E1 -2894.596,E2 -2894.596} C_VEL
LIN {X 0,Y 559.15,Z 174.836,A -85,B 0,C 180,E1 -2897.558,E2 -2897.558} C_VEL
LIN {X 0,Y 559.158,Z 174.831,A -85,B 0,C 180,E1 -2899.838,E2 -2899.838} C_VEL
LIN {X 0,Y 559.134,Z 174.831,A -85,B 0,C 180,E1 -2902.153,E2 -2902.153} C_VEL
LIN {X 0,Y 559.168,Z 174.837,A -85,B 0,C 180,E1 -2905.299,E2 -2905.299} C_VEL
LIN {X 0,Y 559.15,Z 174.832,A -85,B 0,C 180,E1 -2907.714,E2 -2907.714} C_VEL
LIN {X 0,Y 559.144,Z 174.83,A -85,B 0,C 180,E1 -2910.184,E2 -2910.184} C_VEL
LIN {X 0,Y 559.147,Z 174.833,A -85,B 0,C 180,E1 -2912.716,E2 -2912.716} C_VEL
LIN {X 0,Y 559.122,Z 174.839,A -85,B 0,C 180,E1 -2915.325,E2 -2915.325} C_VEL
LIN {X 0,Y 559.125,Z 174.832,A -85,B 0,C 180,E1 -2918.019,E2 -2918.019} C_VEL
LIN {X 0,Y 559.15,Z 174.835,A -85,B 0,C 180,E1 -2920.813,E2 -2920.813} C_VEL
LIN {X 0,Y 559.133,Z 174.832,A -85,B 0,C 180,E1 -2923.735,E2 -2923.735} C_VEL
LIN {X 0,Y 559.136,Z 174.839,A -85,B 0,C 180,E1 -2926.805,E2 -2926.805} C_VEL
LIN {X 0,Y 559.15,Z 174.834,A -85,B 0,C 180,E1 -2929.188,E2 -2929.188} C_VEL
LIN {X 0,Y 559.127,Z 174.832,A -85,B 0,C 180,E1 -2931.983,E2 -2931.983} C_VEL
LIN {X 0,Y 559.126,Z 174.842,A -85,B 0,C 180,E1 -2934.789,E2 -2934.789} C_VEL
LIN {X 0,Y 559.151,Z 174.832,A -85,B 0,C 180,E1 -2937.366,E2 -2937.366} C_VEL
LIN {X 0,Y 559.118,Z 174.837,A -85,B 0,C 180,E1 -2940.149,E2 -2940.149} C_VEL
LIN {X 0,Y 559.157,Z 174.836,A -85,B 0,C 180,E1 -2943.098,E2 -2943.098} C_VEL
LIN {X 0,Y 559.188,Z 175.008,A -85,B 0,C 180,E1 -2945.279,E2 -2945.279} C_VEL
LIN {X 0,Y 560.676,Z 182.426,A -85,B 0,C 180,E1 -2946.213,E2 -2946.213} C_VEL
LIN {X 0,Y 560.3,Z 207.599,A -85,B 0,C 180,E1 -2949.055,E2 -2949.055} C_VEL
LIN {X 0,Y 559.98,Z 231.628,A -85,B 0,C 180,E1 -2951.715,E2 -2951.715} C_VEL
LIN {X 0,Y 559.722,Z 255.6,A -85,B 0,C 180,E1 -2954.339,E2 -2954.339} C_VEL
LIN {X 0,Y 559.622,Z 268.904,A -85,B 0,C 180,E1 -2955.779,E2 -2955.779} C_VEL
LIN {X 0,Y 560.298,Z 276.56,A -85,B 0,C 180,E1 -2955.912,E2 -2955.912} C_VEL
LIN {X 0,Y 560.076,Z 378.978,A -85,B 0,C 180,E1 -2957.246,E2 -2957.246} C_VEL
LIN {X 0,Y 559.949,Z 392.238,A -85,B 0,C 180,E1 -2957.566,E2 -2957.566} C_VEL
LIN {X 0,Y 559.785,Z 405.172,A -85,B 0,C 180,E1 -2958.031,E2 -2958.031} C_VEL
LIN {X 0,Y 559.633,Z 417.856,A -85,B 0,C 180,E1 -2958.664,E2 -2958.664} C_VEL
LIN {X 0,Y 559.446,Z 429.495,A -85,B 0,C 180,E1 -2959.414,E2 -2959.414} C_VEL
LIN {X 0,Y 559.296,Z 439.653,A -85,B 0,C 180,E1 -2960.234,E2 -2960.234} C_VEL
LIN {X 0,Y 559.134,Z 448.791,A -85,B 0,C 180,E1 -2961.143,E2 -2961.143} C_VEL
LIN {X 0,Y 559.009,Z 457.692,A -85,B 0,C 180,E1 -2962.233,E2 -2962.233} C_VEL
LIN {X 0,Y 558.924,Z 463.743,A -85,B 0,C 180,E1 -2963.14,E2 -2963.14} C_VEL
LIN {X 0,Y 558.935,Z 469.682,A -85,B 0,C 180,E1 -2964.227,E2 -2964.227} C_VEL
LIN {X 0,Y 558.826,Z 474.375,A -85,B 0,C 180,E1 -2965.312,E2 -2965.312} C_VEL
LIN {X 0,Y 558.836,Z 477.96,A -85,B 0,C 180,E1 -2966.395,E2 -2966.395} C_VEL
LIN {X 0,Y 558.799,Z 479.808,A -85,B 0,C 180,E1 -2967.117,E2 -2967.117} C_VEL
LIN {X 0,Y 558.745,Z 482.184,A -85,B 0,C 180,E1 -2968.559,E2 -2968.559} C_VEL
LIN {X 0,Y 558.74,Z 483,A -85,B 0,C 180,E1 -2970.001,E2 -2970.001} C_VEL
LIN {X 0,Y 558.745,Z 482.184,A -85,B 0,C 180,E1 -2971.442,E2 -2971.442} C_VEL
LIN {X 0,Y 558.799,Z 479.809,A -85,B 0,C 180,E1 -2972.884,E2 -2972.884} C_VEL
LIN {X 0,Y 558.844,Z 476.894,A -85,B 0,C 180,E1 -2973.967,E2 -2973.967} C_VEL
LIN {X 0,Y 558.798,Z 472.946,A -85,B 0,C 180,E1 -2975.051,E2 -2975.051} C_VEL
LIN {X 0,Y 558.921,Z 467.865,A -85,B 0,C 180,E1 -2976.136,E2 -2976.136} C_VEL
LIN {X 0,Y 558.978,Z 461.464,A -85,B 0,C 180,E1 -2977.223,E2 -2977.223} C_VEL
LIN {X 0,Y 559.099,Z 453.474,A -85,B 0,C 180,E1 -2978.312,E2 -2978.312} C_VEL
LIN {X 0,Y 559.195,Z 445.33,A -85,B 0,C 180,E1 -2979.221,E2 -2979.221} C_VEL
LIN {X 0,Y 559.362,Z 435.393,A -85,B 0,C 180,E1 -2980.131,E2 -2980.131} C_VEL
LIN {X 0,Y 559.538,Z 424.391,A -85,B 0,C 180,E1 -2980.937,E2 -2980.937} C_VEL
LIN {X 0,Y 559.673,Z 412.45,A -85,B 0,C 180,E1 -2981.628,E2 -2981.628} C_VEL
LIN {X 0,Y 559.825,Z 399.757,A -85,B 0,C 180,E1 -2982.185,E2 -2982.185} C_VEL
LIN {X 0,Y 559.987,Z 386.329,A -85,B 0,C 180,E1 -2982.596,E2 -2982.596} C_VEL
LIN {X 0,Y 560.066,Z 373.057,A -85,B 0,C 180,E1 -2982.847,E2 -2982.847} C_VEL
LIN {X 0,Y 560.196,Z 273.574,A -85,B 0,C 180,E1 -2984.129,E2 -2984.129} C_VEL
LIN {X 0,Y 559.603,Z 268.886,A -85,B 0,C 180,E1 -2984.223,E2 -2984.223} C_VEL
LIN {X 0,Y 559.886,Z 240.146,A -85,B 0,C 180,E1 -2987.33,E2 -2987.33} C_VEL
LIN {X 0,Y 560.175,Z 212.24,A -85,B 0,C 180,E1 -2990.375,E2 -2990.375} C_VEL
LIN {X 0,Y 560.466,Z 185.891,A -85,B 0,C 180,E1 -2993.266,E2 -2993.266} C_VEL
LIN {X 0,Y 560.344,Z 180.71,A -85,B 0,C 180,E1 -2993.84,E2 -2993.84} C_VEL
LIN {X 0,Y 559.167,Z 174.943,A -85,B 0,C 180,E1 -2994.553,E2 -2994.553} C_VEL
LIN {X 0,Y 559.138,Z 174.838,A -85,B 0,C 180,E1 -2996.904,E2 -2996.904} C_VEL
LIN {X 0,Y 559.122,Z 174.836,A -85,B 0,C 180,E1 -2999.852,E2 -2999.852} C_VEL
LIN {X 0,Y 559.15,Z 174.833,A -85,B 0,C 180,E1 -3002.716,E2 -3002.716} C_VEL
LIN {X 0,Y 559.124,Z 174.841,A -85,B 0,C 180,E1 -3005.325,E2 -3005.325} C_VEL
LIN {X 0,Y 559.13,Z 174.833,A -85,B 0,C 180,E1 -3008.018,E2 -3008.018} C_VEL
LIN {X 0,Y 559.156,Z 174.835,A -85,B 0,C 180,E1 -3010.813,E2 -3010.813} C_VEL
LIN {X 0,Y 559.138,Z 174.832,A -85,B 0,C 180,E1 -3013.734,E2 -3013.734} C_VEL
LIN {X 0,Y 559.133,Z 174.839,A -85,B 0,C 180,E1 -3016.805,E2 -3016.805} C_VEL
LIN {X 0,Y 559.156,Z 174.834,A -85,B 0,C 180,E1 -3019.187,E2 -3019.187} C_VEL
LIN {X 0,Y 559.131,Z 174.832,A -85,B 0,C 180,E1 -3021.982,E2 -3021.982} C_VEL
LIN {X 0,Y 559.133,Z 174.84,A -85,B 0,C 180,E1 -3024.787,E2 -3024.787} C_VEL
LIN {X 0,Y 559.154,Z 174.831,A -85,B 0,C 180,E1 -3027.365,E2 -3027.365} C_VEL
LIN {X 0,Y 559.144,Z 174.832,A -85,B 0,C 180,E1 -3030.144,E2 -3030.144} C_VEL
LIN {X 0,Y 559.167,Z 174.83,A -85,B 0,C 180,E1 -3033.173,E2 -3033.173} C_VEL
LIN {X 0,Y 559.156,Z 174.829,A -85,B 0,C 180,E1 -3035.495,E2 -3035.495} C_VEL
LIN {X 0,Y 559.173,Z 174.836,A -85,B 0,C 180,E1 -3038.624,E2 -3038.624} C_VEL
LIN {X 0,Y 559.161,Z 174.833,A -85,B 0,C 180,E1 -3040.926,E2 -3040.926} C_VEL
LIN {X 0,Y 559.162,Z 174.831,A -85,B 0,C 180,E1 -3043.947,E2 -3043.947} C_VEL
LIN {X 0,Y 559.166,Z 174.834,A -85,B 0,C 180,E1 -3046.184,E2 -3046.184} C_VEL
LIN {X 0,Y 559.194,Z 174.826,A -85,B 0,C 180,E1 -3049.133,E2 -3049.133} C_VEL
LIN {X 0,Y 559.195,Z 174.83,A -85,B 0,C 180,E1 -3052.053,E2 -3052.053} C_VEL
LIN {X 0,Y 559.247,Z 174.82,A -85,B 0,C 180,E1 -3054.953,E2 -3054.953} C_VEL
LIN {X 0,Y 559.247,Z 174.823,A -85,B 0,C 180,E1 -3057.839,E2 -3057.839} C_VEL
LIN {X 0,Y 559.243,Z 175.009,A -85,B 0,C 180,E1 -3060.315,E2 -3060.315} C_VEL
LIN {X 0,Y 559.246,Z 185.03,A -85,B 0,C 180,E1 -3061.98,E2 -3061.98} C_VEL
LIN {X 0,Y 559.191,Z 194.423,A -85,B 0,C 180,E1 -3063.603,E2 -3063.603} C_VEL
LIN {X 0,Y 559.19,Z 206.905,A -85,B 0,C 180,E1 -3065.77,E2 -3065.77} C_VEL
LIN {X 0,Y 559.073,Z 220.513,A -85,B 0,C 180,E1 -3068.312,E2 -3068.312} C_VEL
LIN {X 0,Y 559.051,Z 223.643,A -85,B 0,C 180,E1 -3068.858,E2 -3068.858} C_VEL
LIN {X 0,Y 559.391,Z 226.368,A -85,B 0,C 180,E1 -3068.944,E2 -3068.944} C_VEL
LIN {X 0,Y 559.713,Z 232.565,A -85,B 0,C 180,E1 -3069.03,E2 -3069.03} C_VEL
LIN {X 0,Y 559.611,Z 299.27,A -85,B 0,C 180,E1 -3069.898,E2 -3069.898} C_VEL
LIN {X 0,Y 559.55,Z 307.747,A -85,B 0,C 180,E1 -3070.082,E2 -3070.082} C_VEL
LIN {X 0,Y 559.487,Z 316.472,A -85,B 0,C 180,E1 -3070.357,E2 -3070.357} C_VEL
LIN {X 0,Y 559.393,Z 324.222,A -85,B 0,C 180,E1 -3070.679,E2 -3070.679} C_VEL
LIN {X 0,Y 559.284,Z 332.431,A -85,B 0,C 180,E1 -3071.112,E2 -3071.112} C_VEL
LIN {X 0,Y 559.221,Z 339.933,A -85,B 0,C 180,E1 -3071.6,E2 -3071.6} C_VEL
LIN {X 0,Y 559.104,Z 348.031,A -85,B 0,C 180,E1 -3072.246,E2 -3072.246} C_VEL
LIN {X 0,Y 559.048,Z 354.698,A -85,B 0,C 180,E1 -3072.893,E2 -3072.893} C_VEL
LIN {X 0,Y 558.973,Z 361.044,A -85,B 0,C 180,E1 -3073.635,E2 -3073.635} C_VEL
LIN {X 0,Y 558.903,Z 366.947,A -85,B 0,C 180,E1 -3074.478,E2 -3074.478} C_VEL
LIN {X 0,Y 558.856,Z 371.992,A -85,B 0,C 180,E1 -3075.379,E2 -3075.379} C_VEL
LIN {X 0,Y 558.818,Z 376.612,A -85,B 0,C 180,E1 -3076.437,E2 -3076.437} C_VEL
LIN {X 0,Y 558.764,Z 379.981,A -85,B 0,C 180,E1 -3077.569,E2 -3077.569} C_VEL
LIN {X 0,Y 558.73,Z 381.603,A -85,B 0,C 180,E1 -3078.358,E2 -3078.358} C_VEL
LIN {X 0,Y 558.057,Z 382.406,A -85,B 0,C 180,E1 -3078.955,E2 -3078.955} C_VEL
LIN {X 0,Y 556.457,Z 382.878,A -85,B 0,C 180,E1 -3079.542,E2 -3079.542} C_VEL
LIN {X 0,Y 552.741,Z 382.733,A -85,B 0,C 180,E1 -3080.715,E2 -3080.715} C_VEL
LIN {X 0,Y 551.732,Z 382.18,A -85,B 0,C 180,E1 -3081.319,E2 -3081.319} C_VEL
LIN {X 0,Y 551.667,Z 381.902,A -85,B 0,C 180,E1 -3081.523,E2 -3081.523} C_VEL
LIN {X 0,Y 551.693,Z 379.249,A -85,B 0,C 180,E1 -3082.863,E2 -3082.863} C_VEL
LIN {X 0,Y 551.739,Z 376.483,A -85,B 0,C 180,E1 -3083.735,E2 -3083.735} C_VEL
LIN {X 0,Y 551.783,Z 371.601,A -85,B 0,C 180,E1 -3084.854,E2 -3084.854} C_VEL
LIN {X 0,Y 551.841,Z 365.885,A -85,B 0,C 180,E1 -3085.861,E2 -3085.861} C_VEL
LIN {X 0,Y 551.924,Z 359.816,A -85,B 0,C 180,E1 -3086.712,E2 -3086.712} C_VEL
LIN {X 0,Y 552.031,Z 351.008,A -85,B 0,C 180,E1 -3087.69,E2 -3087.69} C_VEL
LIN {X 0,Y 552.168,Z 342.828,A -85,B 0,C 180,E1 -3088.398,E2 -3088.398} C_VEL
LIN {X 0,Y 552.304,Z 333.849,A -85,B 0,C 180,E1 -3089.021,E2 -3089.021} C_VEL
LIN {X 0,Y 552.419,Z 324.397,A -85,B 0,C 180,E1 -3089.537,E2 -3089.537} C_VEL
LIN {X 0,Y 552.554,Z 313.01,A -85,B 0,C 180,E1 -3089.997,E2 -3089.997} C_VEL
LIN {X 0,Y 552.62,Z 301.864,A -85,B 0,C 180,E1 -3090.284,E2 -3090.284} C_VEL
LIN {X 0,Y 552.662,Z 272.587,A -85,B 0,C 180,E1 -3090.694,E2 -3090.694} C_VEL
LIN {X 0,Y 552.664,Z 228.414,A -85,B 0,C 180,E1 -3091.27,E2 -3091.27} C_VEL
LIN {X 0,Y 552.059,Z 223.902,A -85,B 0,C 180,E1 -3091.383,E2 -3091.383} C_VEL
LIN {X 0,Y 552.052,Z 217.199,A -85,B 0,C 180,E1 -3092.584,E2 -3092.584} C_VEL
LIN {X 0,Y 552.229,Z 203.398,A -85,B 0,C 180,E1 -3095.199,E2 -3095.199} C_VEL
LIN {X 0,Y 552.318,Z 188.67,A -85,B 0,C 180,E1 -3097.915,E2 -3097.915} C_VEL
LIN {X 0,Y 552.414,Z 178.391,A -85,B 0,C 180,E1 -3099.858,E2 -3099.858} C_VEL
LIN {X 0,Y 552.192,Z 175.76,A -85,B 0,C 180,E1 -3100.411,E2 -3100.411} C_VEL
LIN {X 0,Y 552.09,Z 175.714,A -85,B 0,C 180,E1 -3103.481,E2 -3103.481} C_VEL
LIN {X 0,Y 552.105,Z 175.708,A -85,B 0,C 180,E1 -3106.576,E2 -3106.576} C_VEL
LIN {X 0,Y 552.108,Z 175.713,A -85,B 0,C 180,E1 -3109.519,E2 -3109.519} C_VEL
LIN {X 0,Y 552.091,Z 175.71,A -85,B 0,C 180,E1 -3112.336,E2 -3112.336} C_VEL
LIN {X 0,Y 552.118,Z 175.707,A -85,B 0,C 180,E1 -3115.053,E2 -3115.053} C_VEL
LIN {X 0,Y 552.115,Z 175.714,A -85,B 0,C 180,E1 -3117.681,E2 -3117.681} C_VEL
LIN {X 0,Y 552.11,Z 175.707,A -85,B 0,C 180,E1 -3120.235,E2 -3120.235} C_VEL
LIN {X 0,Y 552.144,Z 175.704,A -85,B 0,C 180,E1 -3122.998,E2 -3122.998} C_VEL
LIN {X 0,Y 552.113,Z 175.711,A -85,B 0,C 180,E1 -3125.161,E2 -3125.161} C_VEL
LIN {X 0,Y 552.124,Z 175.704,A -85,B 0,C 180,E1 -3128.337,E2 -3128.337} C_VEL
LIN {X 0,Y 552.15,Z 175.702,A -85,B 0,C 180,E1 -3130.674,E2 -3130.674} C_VEL
LIN {X 0,Y 552.115,Z 175.709,A -85,B 0,C 180,E1 -3133.737,E2 -3133.737} C_VEL
LIN {X 0,Y 552.134,Z 175.704,A -85,B 0,C 180,E1 -3136.004,E2 -3136.004} C_VEL
LIN {X 0,Y 552.162,Z 175.705,A -85,B 0,C 180,E1 -3138.993,E2 -3138.993} C_VEL
LIN {X 0,Y 552.158,Z 175.701,A -85,B 0,C 180,E1 -3141.951,E2 -3141.951} C_VEL
LIN {X 0,Y 552.228,Z 175.697,A -85,B 0,C 180,E1 -3144.888,E2 -3144.888} C_VEL
LIN {X 0,Y 552.226,Z 175.693,A -85,B 0,C 180,E1 -3147.811,E2 -3147.811} C_VEL
LIN {X 0,Y 552.239,Z 175.694,A -85,B 0,C 180,E1 -3150.729,E2 -3150.729} C_VEL
LIN {X 0,Y 552.202,Z 175.703,A -85,B 0,C 180,E1 -3152.918,E2 -3152.918} C_VEL
LIN {X 0,Y 552.2,Z 175.695,A -85,B 0,C 180,E1 -3155.843,E2 -3155.843} C_VEL
LIN {X 0,Y 552.155,Z 175.708,A -85,B 0,C 180,E1 -3158.785,E2 -3158.785} C_VEL
LIN {X 0,Y 552.159,Z 175.7,A -85,B 0,C 180,E1 -3161.75,E2 -3161.75} C_VEL
LIN {X 0,Y 552.133,Z 175.711,A -85,B 0,C 180,E1 -3164.748,E2 -3164.748} C_VEL
LIN {X 0,Y 552.107,Z 175.707,A -85,B 0,C 180,E1 -3167.788,E2 -3167.788} C_VEL
LIN {X 0,Y 552.127,Z 175.705,A -85,B 0,C 180,E1 -3170.101,E2 -3170.101} C_VEL
LIN {X 0,Y 552.092,Z 175.714,A -85,B 0,C 180,E1 -3172.45,E2 -3172.45} C_VEL
LIN {X 0,Y 552.152,Z 175.702,A -85,B 0,C 180,E1 -3175.35,E2 -3175.35} C_VEL
LIN {X 0,Y 552.122,Z 175.707,A -85,B 0,C 180,E1 -3178.097,E2 -3178.097} C_VEL
LIN {X 0,Y 552.102,Z 175.717,A -85,B 0,C 180,E1 -3180.608,E2 -3180.608} C_VEL
LIN {X 0,Y 552.123,Z 175.706,A -85,B 0,C 180,E1 -3183.184,E2 -3183.184} C_VEL
LIN {X 0,Y 552.107,Z 175.708,A -85,B 0,C 180,E1 -3185.841,E2 -3185.841} C_VEL
LIN {X 0,Y 552.118,Z 175.707,A -85,B 0,C 180,E1 -3189.061,E2 -3189.061} C_VEL
LIN {X 0,Y 552.133,Z 175.703,A -85,B 0,C 180,E1 -3191.444,E2 -3191.444} C_VEL
LIN {X 0,Y 552.089,Z 175.716,A -85,B 0,C 180,E1 -3194.532,E2 -3194.532} C_VEL
LIN {X 0,Y 552.123,Z 175.705,A -85,B 0,C 180,E1 -3197.584,E2 -3197.584} C_VEL
LIN {X 0,Y 552.127,Z 175.711,A -85,B 0,C 180,E1 -3200.473,E2 -3200.473} C_VEL
LIN {X 0,Y 552.106,Z 175.707,A -85,B 0,C 180,E1 -3203.315,E2 -3203.315} C_VEL
LIN {X 0,Y 552.132,Z 175.709,A -85,B 0,C 180,E1 -3205.94,E2 -3205.94} C_VEL
LIN {X 0,Y 552.11,Z 175.71,A -85,B 0,C 180,E1 -3208.54,E2 -3208.54} C_VEL
LIN {X 0,Y 552.118,Z 175.706,A -85,B 0,C 180,E1 -3211.437,E2 -3211.437} C_VEL
LIN {X 0,Y 552.121,Z 175.71,A -85,B 0,C 180,E1 -3214.356,E2 -3214.356} C_VEL
LIN {X 0,Y 552.102,Z 175.708,A -85,B 0,C 180,E1 -3216.758,E2 -3216.758} C_VEL
LIN {X 0,Y 552.118,Z 175.705,A -85,B 0,C 180,E1 -3219.12,E2 -3219.12} C_VEL
LIN {X 0,Y 552.123,Z 175.707,A -85,B 0,C 180,E1 -3221.445,E2 -3221.445} C_VEL
LIN {X 0,Y 552.111,Z 175.713,A -85,B 0,C 180,E1 -3223.738,E2 -3223.738} C_VEL
LIN {X 0,Y 552.127,Z 175.712,A -85,B 0,C 180,E1 -3226.005,E2 -3226.005} C_VEL
LIN {X 0,Y 552.17,Z 175.699,A -85,B 0,C 180,E1 -3228.994,E2 -3228.994} C_VEL
LIN {X 0,Y 552.151,Z 175.708,A -85,B 0,C 180,E1 -3231.952,E2 -3231.952} C_VEL
LIN {X 0,Y 552.221,Z 175.693,A -85,B 0,C 180,E1 -3234.889,E2 -3234.889} C_VEL
LIN {X 0,Y 552.213,Z 175.702,A -85,B 0,C 180,E1 -3237.812,E2 -3237.812} C_VEL
LIN {X 0,Y 552.234,Z 175.691,A -85,B 0,C 180,E1 -3240.73,E2 -3240.73} C_VEL
LIN {X 0,Y 552.198,Z 175.696,A -85,B 0,C 180,E1 -3242.918,E2 -3242.918} C_VEL
LIN {X 0,Y 552.189,Z 175.702,A -85,B 0,C 180,E1 -3245.844,E2 -3245.844} C_VEL
LIN {X 0,Y 552.137,Z 175.703,A -85,B 0,C 180,E1 -3248.786,E2 -3248.786} C_VEL
LIN {X 0,Y 552.155,Z 175.706,A -85,B 0,C 180,E1 -3251.751,E2 -3251.751} C_VEL
LIN {X 0,Y 552.128,Z 175.705,A -85,B 0,C 180,E1 -3254.749,E2 -3254.749} C_VEL
LIN {X 0,Y 552.1,Z 175.711,A -85,B 0,C 180,E1 -3257.789,E2 -3257.789} C_VEL
LIN {X 0,Y 552.119,Z 175.706,A -85,B 0,C 180,E1 -3260.102,E2 -3260.102} C_VEL
LIN {X 0,Y 552.085,Z 175.709,A -85,B 0,C 180,E1 -3262.452,E2 -3262.452} C_VEL
LIN {X 0,Y 552.148,Z 175.71,A -85,B 0,C 180,E1 -3265.351,E2 -3265.351} C_VEL
LIN {X 0,Y 552.09,Z 175.709,A -85,B 0,C 180,E1 -3268.1,E2 -3268.1} C_VEL
LIN {X 0,Y 552.096,Z 175.71,A -85,B 0,C 180,E1 -3270.61,E2 -3270.61} C_VEL
LIN {X 0,Y 552.101,Z 175.717,A -85,B 0,C 180,E1 -3273.187,E2 -3273.187} C_VEL
LIN {X 0,Y 552.08,Z 175.711,A -85,B 0,C 180,E1 -3275.844,E2 -3275.844} C_VEL
LIN {X 0,Y 552.115,Z 175.716,A -85,B 0,C 180,E1 -3279.062,E2 -3279.062} C_VEL
LIN {X 0,Y 552.115,Z 175.709,A -85,B 0,C 180,E1 -3281.447,E2 -3281.447} C_VEL
LIN {X 0,Y 552.087,Z 175.712,A -85,B 0,C 180,E1 -3284.532,E2 -3284.532} C_VEL
LIN {X 0,Y 552.104,Z 175.708,A -85,B 0,C 180,E1 -3287.588,E2 -3287.588} C_VEL
LIN {X 0,Y 552.127,Z 175.707,A -85,B 0,C 180,E1 -3290.474,E2 -3290.474} C_VEL
LIN {X 0,Y 552.096,Z 175.711,A -85,B 0,C 180,E1 -3293.319,E2 -3293.319} C_VEL
LIN {X 0,Y 552.122,Z 175.706,A -85,B 0,C 180,E1 -3295.94,E2 -3295.94} C_VEL
LIN {X 0,Y 552.118,Z 175.713,A -85,B 0,C 180,E1 -3298.542,E2 -3298.542} C_VEL
LIN {X 0,Y 552.101,Z 175.71,A -85,B 0,C 180,E1 -3301.443,E2 -3301.443} C_VEL
LIN {X 0,Y 552.104,Z 175.712,A -85,B 0,C 180,E1 -3303.543,E2 -3303.543} C_VEL
LIN {X 0,Y 552.155,Z 175.894,A -85,B 0,C 180,E1 -3305.089,E2 -3305.089} C_VEL
LIN {X 0,Y 553.826,Z 184.429,A -85,B 0,C 180,E1 -3306.175,E2 -3306.175} C_VEL
LIN {X 0,Y 553.381,Z 210.669,A -85,B 0,C 180,E1 -3309.17,E2 -3309.17} C_VEL
LIN {X 0,Y 552.943,Z 238.071,A -85,B 0,C 180,E1 -3312.24,E2 -3312.24} C_VEL
LIN {X 0,Y 552.609,Z 265.421,A -85,B 0,C 180,E1 -3315.265,E2 -3315.265} C_VEL
LIN {X 0,Y 552.622,Z 268.875,A -85,B 0,C 180,E1 -3315.618,E2 -3315.618} C_VEL
LIN {X 0,Y 553.391,Z 277.159,A -85,B 0,C 180,E1 -3315.756,E2 -3315.756} C_VEL
LIN {X 0,Y 553.139,Z 378.697,A -85,B 0,C 180,E1 -3317.084,E2 -3317.084} C_VEL
LIN {X 0,Y 553.03,Z 392.137,A -85,B 0,C 180,E1 -3317.408,E2 -3317.408} C_VEL
LIN {X 0,Y 552.812,Z 404.37,A -85,B 0,C 180,E1 -3317.845,E2 -3317.845} C_VEL
LIN {X 0,Y 552.689,Z 416.677,A -85,B 0,C 180,E1 -3318.45,E2 -3318.45} C_VEL
LIN {X 0,Y 552.49,Z 428.201,A -85,B 0,C 180,E1 -3319.186,E2 -3319.186} C_VEL
LIN {X 0,Y 552.276,Z 438.612,A -85,B 0,C 180,E1 -3320.016,E2 -3320.016} C_VEL
LIN {X 0,Y 552.126,Z 447.119,A -85,B 0,C 180,E1 -3320.845,E2 -3320.845} C_VEL
LIN {X 0,Y 552.013,Z 454.965,A -85,B 0,C 180,E1 -3321.766,E2 -3321.766} C_VEL
LIN {X 0,Y 551.889,Z 462.625,A -85,B 0,C 180,E1 -3322.868,E2 -3322.868} C_VEL
LIN {X 0,Y 551.867,Z 469.682,A -85,B 0,C 180,E1 -3324.153,E2 -3324.153} C_VEL
LIN {X 0,Y 551.725,Z 474.375,A -85,B 0,C 180,E1 -3325.251,E2 -3325.251} C_VEL
LIN {X 0,Y 551.75,Z 477.959,A -85,B 0,C 180,E1 -3326.349,E2 -3326.349} C_VEL
LIN {X 0,Y 551.723,Z 479.808,A -85,B 0,C 180,E1 -3327.08,E2 -3327.08} C_VEL
LIN {X 0,Y 551.645,Z 482.183,A -85,B 0,C 180,E1 -3328.54,E2 -3328.54} C_VEL
LIN {X 0,Y 551.64,Z 483,A -85,B 0,C 180,E1 -3330.001,E2 -3330.001} C_VEL
LIN {X 0,Y 551.645,Z 482.183,A -85,B 0,C 180,E1 -3331.461,E2 -3331.461} C_VEL
LIN {X 0,Y 551.724,Z 479.809,A -85,B 0,C 180,E1 -3332.921,E2 -3332.921} C_VEL
LIN {X 0,Y 551.764,Z 476.894,A -85,B 0,C 180,E1 -3334.018,E2 -3334.018} C_VEL
LIN {X 0,Y 551.724,Z 472.946,A -85,B 0,C 180,E1 -3335.116,E2 -3335.116} C_VEL
LIN {X 0,Y 551.803,Z 467.19,A -85,B 0,C 180,E1 -3336.341,E2 -3336.341} C_VEL
LIN {X 0,Y 551.927,Z 460.232,A -85,B 0,C 180,E1 -3337.5,E2 -3337.5} C_VEL
LIN {X 0,Y 552.083,Z 451.988,A -85,B 0,C 180,E1 -3338.603,E2 -3338.603} C_VEL
LIN {X 0,Y 552.201,Z 443.535,A -85,B 0,C 180,E1 -3339.524,E2 -3339.524} C_VEL
LIN {X 0,Y 552.425,Z 433.086,A -85,B 0,C 180,E1 -3340.445,E2 -3340.445} C_VEL
LIN {X 0,Y 552.614,Z 421.171,A -85,B 0,C 180,E1 -3341.286,E2 -3341.286} C_VEL
LIN {X 0,Y 552.807,Z 409.477,A -85,B 0,C 180,E1 -3341.923,E2 -3341.923} C_VEL
LIN {X 0,Y 552.943,Z 398.409,A -85,B 0,C 180,E1 -3342.386,E2 -3342.386} C_VEL
LIN {X 0,Y 553.059,Z 385.214,A -85,B 0,C 180,E1 -3342.779,E2 -3342.779} C_VEL
LIN {X 0,Y 553.148,Z 372.571,A -85,B 0,C 180,E1 -3343.011,E2 -3343.011} C_VEL
LIN {X 0,Y 553.24,Z 273.996,A -85,B 0,C 180,E1 -3344.287,E2 -3344.287} C_VEL
LIN {X 0,Y 552.605,Z 268.751,A -85,B 0,C 180,E1 -3344.383,E2 -3344.383} C_VEL
LIN {X 0,Y 552.908,Z 239.34,A -85,B 0,C 180,E1 -3347.574,E2 -3347.574} C_VEL
LIN {X 0,Y 553.246,Z 209.847,A -85,B 0,C 180,E1 -3350.836,E2 -3350.836} C_VEL
LIN {X 0,Y 553.566,Z 183.407,A -85,B 0,C 180,E1 -3353.764,E2 -3353.764} C_VEL
LIN {X 0,Y 552.169,Z 175.847,A -85,B 0,C 180,E1 -3354.686,E2 -3354.686} C_VEL
LIN {X 0,Y 552.083,Z 175.719,A -85,B 0,C 180,E1 -3357.276,E2 -3357.276} C_VEL
LIN {X 0,Y 552.098,Z 175.71,A -85,B 0,C 180,E1 -3360.047,E2 -3360.047} C_VEL
LIN {X 0,Y 552.11,Z 175.712,A -85,B 0,C 180,E1 -3362.845,E2 -3362.845} C_VEL
LIN {X 0,Y 552.072,Z 175.718,A -85,B 0,C 180,E1 -3365.438,E2 -3365.438} C_VEL
LIN {X 0,Y 552.094,Z 175.71,A -85,B 0,C 180,E1 -3367.885,E2 -3367.885} C_VEL
LIN {X 0,Y 552.109,Z 175.709,A -85,B 0,C 180,E1 -3370.481,E2 -3370.481} C_VEL
LIN {X 0,Y 552.095,Z 175.712,A -85,B 0,C 180,E1 -3373.481,E2 -3373.481} C_VEL
LIN {X 0,Y 552.074,Z 175.715,A -85,B 0,C 180,E1 -3376.573,E2 -3376.573} C_VEL
LIN {X 0,Y 552.109,Z 175.708,A -85,B 0,C 180,E1 -3379.518,E2 -3379.518} C_VEL
LIN {X 0,Y 552.092,Z 175.711,A -85,B 0,C 180,E1 -3382.336,E2 -3382.336} C_VEL
LIN {X 0,Y 552.084,Z 175.716,A -85,B 0,C 180,E1 -3385.051,E2 -3385.051} C_VEL
LIN {X 0,Y 552.115,Z 175.706,A -85,B 0,C 180,E1 -3387.681,E2 -3387.681} C_VEL
LIN {X 0,Y 552.108,Z 175.71,A -85,B 0,C 180,E1 -3390.234,E2 -3390.234} C_VEL
LIN {X 0,Y 552.135,Z 175.709,A -85,B 0,C 180,E1 -3393.001,E2 -3393.001} C_VEL
LIN {X 0,Y 552.114,Z 175.709,A -85,B 0,C 180,E1 -3395.161,E2 -3395.161} C_VEL
LIN {X 0,Y 552.128,Z 175.71,A -85,B 0,C 180,E1 -3398.337,E2 -3398.337} C_VEL
LIN {X 0,Y 552.151,Z 175.709,A -85,B 0,C 180,E1 -3400.674,E2 -3400.674} C_VEL
LIN {X 0,Y 552.113,Z 175.708,A -85,B 0,C 180,E1 -3403.737,E2 -3403.737} C_VEL
LIN {X 0,Y 552.132,Z 175.708,A -85,B 0,C 180,E1 -3406.004,E2 -3406.004} C_VEL
LIN {X 0,Y 552.162,Z 175.703,A -85,B 0,C 180,E1 -3408.993,E2 -3408.993} C_VEL
LIN {X 0,Y 552.15,Z 175.706,A -85,B 0,C 180,E1 -3411.951,E2 -3411.951} C_VEL
LIN {X 0,Y 552.222,Z 175.696,A -85,B 0,C 180,E1 -3414.889,E2 -3414.889} C_VEL
LIN {X 0,Y 552.219,Z 175.698,A -85,B 0,C 180,E1 -3417.812,E2 -3417.812} C_VEL
LIN {X 0,Y 552.195,Z 175.8,A -85,B 0,C 180,E1 -3420.341,E2 -3420.341} C_VEL
LIN {X 0,Y 552.162,Z 191.219,A -85,B 0,C 180,E1 -3422.918,E2 -3422.918} C_VEL
LIN {X 0,Y 552.16,Z 206.278,A -85,B 0,C 180,E1 -3425.478,E2 -3425.478} C_VEL
LIN {X 0,Y 552.032,Z 220.09,A -85,B 0,C 180,E1 -3428.05,E2 -3428.05} C_VEL
LIN {X 0,Y 552.072,Z 224.133,A -85,B 0,C 180,E1 -3428.717,E2 -3428.717} C_VEL
LIN {X 0,Y 552.781,Z 230.52,A -85,B 0,C 180,E1 -3428.844,E2 -3428.844} C_VEL
LIN {X 0,Y 552.617,Z 300.03,A -85,B 0,C 180,E1 -3429.77,E2 -3429.77} C_VEL
LIN {X 0,Y 552.555,Z 309.161,A -85,B 0,C 180,E1 -3429.979,E2 -3429.979} C_VEL
LIN {X 0,Y 552.504,Z 318.749,A -85,B 0,C 180,E1 -3430.304,E2 -3430.304} C_VEL
LIN {X 0,Y 552.383,Z 329.715,A -85,B 0,C 180,E1 -3430.816,E2 -3430.816} C_VEL
LIN {X 0,Y 552.205,Z 340.068,A -85,B 0,C 180,E1 -3431.481,E2 -3431.481} C_VEL
LIN {X 0,Y 552.096,Z 347.99,A -85,B 0,C 180,E1 -3432.124,E2 -3432.124} C_VEL
LIN {X 0,Y 552.017,Z 353.784,A -85,B 0,C 180,E1 -3432.686,E2 -3432.686} C_VEL
LIN {X 0,Y 551.901,Z 360.249,A -85,B 0,C 180,E1 -3433.438,E2 -3433.438} C_VEL
LIN {X 0,Y 551.864,Z 366.131,A -85,B 0,C 180,E1 -3434.275,E2 -3434.275} C_VEL
LIN {X 0,Y 551.813,Z 371.057,A -85,B 0,C 180,E1 -3435.134,E2 -3435.134} C_VEL
LIN {X 0,Y 551.735,Z 374.596,A -85,B 0,C 180,E1 -3435.894,E2 -3435.894} C_VEL
LIN {X 0,Y 551.719,Z 377.46,A -85,B 0,C 180,E1 -3436.655,E2 -3436.655} C_VEL
LIN {X 0,Y 551.712,Z 379.11,A -85,B 0,C 180,E1 -3437.179,E2 -3437.179} C_VEL
LIN {X 0,Y 551.641,Z 381.541,A -85,B 0,C 180,E1 -3438.359,E2 -3438.359} C_VEL
LIN {X 0,Y 551.678,Z 382.782,A -85,B 0,C 180,E1 -3439.488,E2 -3439.488} C_VEL
LIN {X 0,Y 551.639,Z 382.988,A -85,B 0,C 180,E1 -3440.119,E2 -3440.119} C_VEL
LIN {X 0,Y 551.642,Z 382.651,A -85,B 0,C 180,E1 -3440.899,E2 -3440.899} C_VEL
LIN {X 0,Y 551.667,Z 381.902,A -85,B 0,C 180,E1 -3441.523,E2 -3441.523} C_VEL
LIN {X 0,Y 551.045,Z 381.021,A -85,B 0,C 180,E1 -3442.127,E2 -3442.127} C_VEL
LIN {X 0,Y 548.21,Z 378.914,A -85,B 0,C 180,E1 -3443.093,E2 -3443.093} C_VEL
LIN {X 0,Y 545.353,Z 375.915,A -85,B 0,C 180,E1 -3444.042,E2 -3444.042} C_VEL
LIN {X 0,Y 544.71,Z 373.579,A -85,B 0,C 180,E1 -3444.613,E2 -3444.613} C_VEL
LIN {X 0,Y 544.806,Z 367.993,A -85,B 0,C 180,E1 -3445.686,E2 -3445.686} C_VEL
LIN {X 0,Y 544.884,Z 361.642,A -85,B 0,C 180,E1 -3446.629,E2 -3446.629} C_VEL
LIN {X 0,Y 544.974,Z 355.592,A -85,B 0,C 180,E1 -3447.361,E2 -3447.361} C_VEL
LIN {X 0,Y 545.058,Z 348.46,A -85,B 0,C 180,E1 -3448.075,E2 -3448.075} C_VEL
LIN {X 0,Y 545.234,Z 339.836,A -85,B 0,C 180,E1 -3448.776,E2 -3448.776} C_VEL
LIN {X 0,Y 545.396,Z 328.599,A -85,B 0,C 180,E1 -3449.477,E2 -3449.477} C_VEL
LIN {X 0,Y 545.542,Z 318.331,A -85,B 0,C 180,E1 -3449.947,E2 -3449.947} C_VEL
LIN {X 0,Y 545.626,Z 307.546,A -85,B 0,C 180,E1 -3450.299,E2 -3450.299} C_VEL
LIN {X 0,Y 545.676,Z 296.38,A -85,B 0,C 180,E1 -3450.524,E2 -3450.524} C_VEL
LIN {X 0,Y 545.691,Z 228.674,A -85,B 0,C 180,E1 -3451.429,E2 -3451.429} C_VEL
LIN {X 0,Y 545.034,Z 224.097,A -85,B 0,C 180,E1 -3451.545,E2 -3451.545} C_VEL
LIN {X 0,Y 545.058,Z 215.71,A -85,B 0,C 180,E1 -3453.059,E2 -3453.059} C_VEL
LIN {X 0,Y 545.197,Z 203.122,A -85,B 0,C 180,E1 -3455.456,E2 -3455.456} C_VEL
LIN {X 0,Y 545.323,Z 188.354,A -85,B 0,C 180,E1 -3458.214,E2 -3458.214} C_VEL
LIN {X 0,Y 545.341,Z 178.307,A -85,B 0,C 180,E1 -3460.118,E2 -3460.118} C_VEL
LIN {X 0,Y 545.151,Z 176.605,A -85,B 0,C 180,E1 -3460.503,E2 -3460.503} C_VEL
LIN {X 0,Y 545.048,Z 176.596,A -85,B 0,C 180,E1 -3463.773,E2 -3463.773} C_VEL
LIN {X 0,Y 545.077,Z 176.584,A -85,B 0,C 180,E1 -3466.893,E2 -3466.893} C_VEL
LIN {X 0,Y 545.064,Z 176.591,A -85,B 0,C 180,E1 -3469.857,E2 -3469.857} C_VEL
LIN {X 0,Y 545.072,Z 176.585,A -85,B 0,C 180,E1 -3473.073,E2 -3473.073} C_VEL
LIN {X 0,Y 545.081,Z 176.592,A -85,B 0,C 180,E1 -3475.606,E2 -3475.606} C_VEL
LIN {X 0,Y 545.056,Z 176.586,A -85,B 0,C 180,E1 -3478.321,E2 -3478.321} C_VEL
LIN {X 0,Y 545.088,Z 176.586,A -85,B 0,C 180,E1 -3481.251,E2 -3481.251} C_VEL
LIN {X 0,Y 545.088,Z 176.583,A -85,B 0,C 180,E1 -3484,E2 -3484} C_VEL
LIN {X 0,Y 545.08,Z 176.582,A -85,B 0,C 180,E1 -3486.44,E2 -3486.44} C_VEL
LIN {X 0,Y 545.091,Z 176.587,A -85,B 0,C 180,E1 -3489.627,E2 -3489.627} C_VEL
LIN {X 0,Y 545.093,Z 176.582,A -85,B 0,C 180,E1 -3492.75,E2 -3492.75} C_VEL
LIN {X 0,Y 545.093,Z 176.583,A -85,B 0,C 180,E1 -3495.82,E2 -3495.82} C_VEL
LIN {X 0,Y 545.117,Z 176.581,A -85,B 0,C 180,E1 -3498.849,E2 -3498.849} C_VEL
LIN {X 0,Y 545.128,Z 176.577,A -85,B 0,C 180,E1 -3501.847,E2 -3501.847} C_VEL
LIN {X 0,Y 545.205,Z 176.571,A -85,B 0,C 180,E1 -3504.822,E2 -3504.822} C_VEL
LIN {X 0,Y 545.197,Z 176.568,A -85,B 0,C 180,E1 -3507.783,E2 -3507.783} C_VEL
LIN {X 0,Y 545.21,Z 176.57,A -85,B 0,C 180,E1 -3510.738,E2 -3510.738} C_VEL
LIN {X 0,Y 545.169,Z 176.579,A -85,B 0,C 180,E1 -3512.955,E2 -3512.955} C_VEL
LIN {X 0,Y 545.17,Z 176.571,A -85,B 0,C 180,E1 -3515.919,E2 -3515.919} C_VEL
LIN {X 0,Y 545.115,Z 176.587,A -85,B 0,C 180,E1 -3518.899,E2 -3518.899} C_VEL
LIN {X 0,Y 545.132,Z 176.576,A -85,B 0,C 180,E1 -3521.904,E2 -3521.904} C_VEL
LIN {X 0,Y 545.082,Z 176.59,A -85,B 0,C 180,E1 -3524.943,E2 -3524.943} C_VEL
LIN {X 0,Y 545.075,Z 176.583,A -85,B 0,C 180,E1 -3528.025,E2 -3528.025} C_VEL
LIN {X 0,Y 545.091,Z 176.584,A -85,B 0,C 180,E1 -3530.371,E2 -3530.371} C_VEL
LIN {X 0,Y 545.087,Z 176.581,A -85,B 0,C 180,E1 -3533.558,E2 -3533.558} C_VEL
LIN {X 0,Y 545.084,Z 176.582,A -85,B 0,C 180,E1 -3535.999,E2 -3535.999} C_VEL
LIN {X 0,Y 545.085,Z 176.589,A -85,B 0,C 180,E1 -3538.748,E2 -3538.748} C_VEL
LIN {X 0,Y 545.072,Z 176.583,A -85,B 0,C 180,E1 -3541.682,E2 -3541.682} C_VEL
LIN {X 0,Y 545.079,Z 176.592,A -85,B 0,C 180,E1 -3544.562,E2 -3544.562} C_VEL
LIN {X 0,Y 545.035,Z 176.588,A -85,B 0,C 180,E1 -3547.303,E2 -3547.303} C_VEL
LIN {X 0,Y 545.085,Z 176.586,A -85,B 0,C 180,E1 -3550.14,E2 -3550.14} C_VEL
LIN {X 0,Y 545.079,Z 176.583,A -85,B 0,C 180,E1 -3553.105,E2 -3553.105} C_VEL
LIN {X 0,Y 545.049,Z 176.593,A -85,B 0,C 180,E1 -3556.225,E2 -3556.225} C_VEL
LIN {X 0,Y 545.093,Z 176.582,A -85,B 0,C 180,E1 -3558.887,E2 -3558.887} C_VEL
LIN {X 0,Y 545.046,Z 176.589,A -85,B 0,C 180,E1 -3561.763,E2 -3561.763} C_VEL
LIN {X 0,Y 545.057,Z 176.59,A -85,B 0,C 180,E1 -3564.534,E2 -3564.534} C_VEL
LIN {X 0,Y 545.075,Z 176.583,A -85,B 0,C 180,E1 -3567.212,E2 -3567.212} C_VEL
LIN {X 0,Y 545.093,Z 176.585,A -85,B 0,C 180,E1 -3569.813,E2 -3569.813} C_VEL
LIN {X 0,Y 545.087,Z 176.582,A -85,B 0,C 180,E1 -3572.826,E2 -3572.826} C_VEL
LIN {X 0,Y 545.044,Z 176.59,A -85,B 0,C 180,E1 -3575.631,E2 -3575.631} C_VEL
LIN {X 0,Y 545.061,Z 176.585,A -85,B 0,C 180,E1 -3578.837,E2 -3578.837} C_VEL
LIN {X 0,Y 545.076,Z 176.583,A -85,B 0,C 180,E1 -3581.196,E2 -3581.196} C_VEL
LIN {X 0,Y 545.067,Z 176.587,A -85,B 0,C 180,E1 -3583.521,E2 -3583.521} C_VEL
LIN {X 0,Y 545.086,Z 176.59,A -85,B 0,C 180,E1 -3585.82,E2 -3585.82} C_VEL
LIN {X 0,Y 545.124,Z 176.576,A -85,B 0,C 180,E1 -3588.85,E2 -3588.85} C_VEL
LIN {X 0,Y 545.121,Z 176.586,A -85,B 0,C 180,E1 -3591.847,E2 -3591.847} C_VEL
LIN {X 0,Y 545.196,Z 176.567,A -85,B 0,C 180,E1 -3594.823,E2 -3594.823} C_VEL
LIN {X 0,Y 545.185,Z 176.577,A -85,B 0,C 180,E1 -3597.784,E2 -3597.784} C_VEL
LIN {X 0,Y 545.204,Z 176.567,A -85,B 0,C 180,E1 -3600.739,E2 -3600.739} C_VEL
LIN {X 0,Y 545.164,Z 176.572,A -85,B 0,C 180,E1 -3602.956,E2 -3602.956} C_VEL
LIN {X 0,Y 545.161,Z 176.576,A -85,B 0,C 180,E1 -3605.92,E2 -3605.92} C_VEL
LIN {X 0,Y 545.1,Z 176.581,A -85,B 0,C 180,E1 -3608.901,E2 -3608.901} C_VEL
LIN {X 0,Y 545.127,Z 176.58,A -85,B 0,C 180,E1 -3611.905,E2 -3611.905} C_VEL
LIN {X 0,Y 545.077,Z 176.585,A -85,B 0,C 180,E1 -3614.944,E2 -3614.944} C_VEL
LIN {X 0,Y 545.068,Z 176.585,A -85,B 0,C 180,E1 -3618.026,E2 -3618.026} C_VEL
LIN {X 0,Y 545.085,Z 176.581,A -85,B 0,C 180,E1 -3620.373,E2 -3620.373} C_VEL
LIN {X 0,Y 545.073,Z 176.588,A -85,B 0,C 180,E1 -3623.56,E2 -3623.56} C_VEL
LIN {X 0,Y 545.071,Z 176.584,A -85,B 0,C 180,E1 -3626.001,E2 -3626.001} C_VEL
LIN {X 0,Y 545.068,Z 176.586,A -85,B 0,C 180,E1 -3628.746,E2 -3628.746} C_VEL
LIN {X 0,Y 545.052,Z 176.588,A -85,B 0,C 180,E1 -3631.68,E2 -3631.68} C_VEL
LIN {X 0,Y 545.054,Z 176.587,A -85,B 0,C 180,E1 -3634.565,E2 -3634.565} C_VEL
LIN {X 0,Y 545.03,Z 176.594,A -85,B 0,C 180,E1 -3637.305,E2 -3637.305} C_VEL
LIN {X 0,Y 545.06,Z 176.585,A -85,B 0,C 180,E1 -3640.144,E2 -3640.144} C_VEL
LIN {X 0,Y 545.074,Z 176.591,A -85,B 0,C 180,E1 -3643.107,E2 -3643.107} C_VEL
LIN {X 0,Y 545.045,Z 176.587,A -85,B 0,C 180,E1 -3646.227,E2 -3646.227} C_VEL
LIN {X 0,Y 545.067,Z 176.593,A -85,B 0,C 180,E1 -3648.885,E2 -3648.885} C_VEL
LIN {X 0,Y 545.078,Z 176.591,A -85,B 0,C 180,E1 -3650.819,E2 -3650.819} C_VEL
LIN {X 0,Y 545.031,Z 176.588,A -85,B 0,C 180,E1 -3653.62,E2 -3653.62} C_VEL
LIN {X 0,Y 545.061,Z 176.588,A -85,B 0,C 180,E1 -3656.329,E2 -3656.329} C_VEL
LIN {X 0,Y 545.06,Z 176.593,A -85,B 0,C 180,E1 -3658.953,E2 -3658.953} C_VEL
LIN {X 0,Y 545.079,Z 176.585,A -85,B 0,C 180,E1 -3661.507,E2 -3661.507} C_VEL
LIN {X 0,Y 545.06,Z 176.591,A -85,B 0,C 180,E1 -3663.999,E2 -3663.999} C_VEL
LIN {X 0,Y 545.108,Z 176.853,A -85,B 0,C 180,E1 -3664.91,E2 -3664.91} C_VEL
LIN {X 0,Y 546.942,Z 185.475,A -85,B 0,C 180,E1 -3666.023,E2 -3666.023} C_VEL
LIN {X 0,Y 546.443,Z 210.297,A -85,B 0,C 180,E1 -3668.893,E2 -3668.893} C_VEL
LIN {X 0,Y 546.01,Z 235.911,A -85,B 0,C 180,E1 -3671.813,E2 -3671.813} C_VEL
LIN {X 0,Y 545.63,Z 261.548,A -85,B 0,C 180,E1 -3674.691,E2 -3674.691} C_VEL
LIN {X 0,Y 545.605,Z 268.686,A -85,B 0,C 180,E1 -3675.454,E2 -3675.454} C_VEL
LIN {X 0,Y 546.471,Z 277.032,A -85,B 0,C 180,E1 -3675.597,E2 -3675.597} C_VEL
LIN {X 0,Y 546.166,Z 378.261,A -85,B 0,C 180,E1 -3676.939,E2 -3676.939} C_VEL
LIN {X 0,Y 546.031,Z 391.675,A -85,B 0,C 180,E1 -3677.267,E2 -3677.267} C_VEL
LIN {X 0,Y 545.805,Z 404.504,A -85,B 0,C 180,E1 -3677.734,E2 -3677.734} C_VEL
LIN {X 0,Y 545.674,Z 416.658,A -85,B 0,C 180,E1 -3678.341,E2 -3678.341} C_VEL
LIN {X 0,Y 545.452,Z 428.979,A -85,B 0,C 180,E1 -3679.139,E2 -3679.139} C_VEL
LIN {X 0,Y 545.236,Z 439.318,A -85,B 0,C 180,E1 -3679.979,E2 -3679.979} C_VEL
LIN {X 0,Y 545.054,Z 448.61,A -85,B 0,C 180,E1 -3680.913,E2 -3680.913} C_VEL
LIN {X 0,Y 544.916,Z 457.652,A -85,B 0,C 180,E1 -3682.031,E2 -3682.031} C_VEL
LIN {X 0,Y 544.785,Z 464.852,A -85,B 0,C 180,E1 -3683.147,E2 -3683.147} C_VEL
LIN {X 0,Y 544.741,Z 471.368,A -85,B 0,C 180,E1 -3684.448,E2 -3684.448} C_VEL
LIN {X 0,Y 544.66,Z 475.678,A -85,B 0,C 180,E1 -3685.56,E2 -3685.56} C_VEL
LIN {X 0,Y 544.669,Z 477.959,A -85,B 0,C 180,E1 -3686.301,E2 -3686.301} C_VEL
LIN {X 0,Y 544.65,Z 479.808,A -85,B 0,C 180,E1 -3687.042,E2 -3687.042} C_VEL
LIN {X 0,Y 544.546,Z 482.182,A -85,B 0,C 180,E1 -3688.521,E2 -3688.521} C_VEL
LIN {X 0,Y 544.541,Z 483,A -85,B 0,C 180,E1 -3690.001,E2 -3690.001} C_VEL
LIN {X 0,Y 544.546,Z 482.183,A -85,B 0,C 180,E1 -3691.48,E2 -3691.48} C_VEL
LIN {X 0,Y 544.651,Z 479.809,A -85,B 0,C 180,E1 -3692.959,E2 -3692.959} C_VEL
LIN {X 0,Y 544.684,Z 476.894,A -85,B 0,C 180,E1 -3694.07,E2 -3694.07} C_VEL
LIN {X 0,Y 544.654,Z 472.946,A -85,B 0,C 180,E1 -3695.183,E2 -3695.183} C_VEL
LIN {X 0,Y 544.74,Z 467.705,A -85,B 0,C 180,E1 -3696.328,E2 -3696.328} C_VEL
LIN {X 0,Y 544.837,Z 461.453,A -85,B 0,C 180,E1 -3697.412,E2 -3697.412} C_VEL
LIN {X 0,Y 545.007,Z 453.376,A -85,B 0,C 180,E1 -3698.529,E2 -3698.529} C_VEL
LIN {X 0,Y 545.114,Z 445.075,A -85,B 0,C 180,E1 -3699.462,E2 -3699.462} C_VEL
LIN {X 0,Y 545.355,Z 434.958,A -85,B 0,C 180,E1 -3700.395,E2 -3700.395} C_VEL
LIN {X 0,Y 545.529,Z 423.926,A -85,B 0,C 180,E1 -3701.209,E2 -3701.209} C_VEL
LIN {X 0,Y 545.695,Z 412.266,A -85,B 0,C 180,E1 -3701.892,E2 -3701.892} C_VEL
LIN {X 0,Y 545.883,Z 399.765,A -85,B 0,C 180,E1 -3702.454,E2 -3702.454} C_VEL
LIN {X 0,Y 546.048,Z 386.43,A -85,B 0,C 180,E1 -3702.875,E2 -3702.875} C_VEL
LIN {X 0,Y 546.166,Z 373.484,A -85,B 0,C 180,E1 -3703.133,E2 -3703.133} C_VEL
LIN {X 0,Y 546.332,Z 274.819,A -85,B 0,C 180,E1 -3704.432,E2 -3704.432} C_VEL
LIN {X 0,Y 545.572,Z 268.426,A -85,B 0,C 180,E1 -3704.548,E2 -3704.548} C_VEL
LIN {X 0,Y 545.886,Z 240.734,A -85,B 0,C 180,E1 -3707.58,E2 -3707.58} C_VEL
LIN {X 0,Y 546.27,Z 212.678,A -85,B 0,C 180,E1 -3710.72,E2 -3710.72} C_VEL
LIN {X 0,Y 546.628,Z 185.263,A -85,B 0,C 180,E1 -3713.786,E2 -3713.786} C_VEL
LIN {X 0,Y 545.114,Z 176.712,A -85,B 0,C 180,E1 -3714.849,E2 -3714.849} C_VEL
LIN {X 0,Y 545.043,Z 176.594,A -85,B 0,C 180,E1 -3717.659,E2 -3717.659} C_VEL
LIN {X 0,Y 545.047,Z 176.589,A -85,B 0,C 180,E1 -3720.24,E2 -3720.24} C_VEL
LIN {X 0,Y 545.073,Z 176.592,A -85,B 0,C 180,E1 -3723.061,E2 -3723.061} C_VEL
LIN {X 0,Y 545.027,Z 176.593,A -85,B 0,C 180,E1 -3725.671,E2 -3725.671} C_VEL
LIN {X 0,Y 545.05,Z 176.587,A -85,B 0,C 180,E1 -3728.238,E2 -3728.238} C_VEL
LIN {X 0,Y 545.031,Z 176.597,A -85,B 0,C 180,E1 -3731.119,E2 -3731.119} C_VEL
LIN {X 0,Y 545.051,Z 176.587,A -85,B 0,C 180,E1 -3734.13,E2 -3734.13} C_VEL
LIN {X 0,Y 545.025,Z 176.597,A -85,B 0,C 180,E1 -3736.888,E2 -3736.888} C_VEL
LIN {X 0,Y 545.081,Z 176.583,A -85,B 0,C 180,E1 -3739.527,E2 -3739.527} C_VEL
LIN {X 0,Y 545.049,Z 176.586,A -85,B 0,C 180,E1 -3741.864,E2 -3741.864} C_VEL
LIN {X 0,Y 545.037,Z 176.593,A -85,B 0,C 180,E1 -3744.531,E2 -3744.531} C_VEL
LIN {X 0,Y 545.066,Z 176.588,A -85,B 0,C 180,E1 -3747.211,E2 -3747.211} C_VEL
LIN {X 0,Y 545.063,Z 176.585,A -85,B 0,C 180,E1 -3749.81,E2 -3749.81} C_VEL
LIN {X 0,Y 545.081,Z 176.59,A -85,B 0,C 180,E1 -3752.829,E2 -3752.829} C_VEL
LIN {X 0,Y 545.05,Z 176.586,A -85,B 0,C 180,E1 -3755.63,E2 -3755.63} C_VEL
LIN {X 0,Y 545.066,Z 176.59,A -85,B 0,C 180,E1 -3758.836,E2 -3758.836} C_VEL
LIN {X 0,Y 545.057,Z 176.587,A -85,B 0,C 180,E1 -3761.194,E2 -3761.194} C_VEL
LIN {X 0,Y 545.064,Z 176.585,A -85,B 0,C 180,E1 -3763.521,E2 -3763.521} C_VEL
LIN {X 0,Y 545.093,Z 176.583,A -85,B 0,C 180,E1 -3765.82,E2 -3765.82} C_VEL
LIN {X 0,Y 545.118,Z 176.582,A -85,B 0,C 180,E1 -3768.849,E2 -3768.849} C_VEL
LIN {X 0,Y 545.098,Z 176.583,A -85,B 0,C 180,E1 -3771.846,E2 -3771.846} C_VEL
LIN {X 0,Y 545.198,Z 176.572,A -85,B 0,C 180,E1 -3774.823,E2 -3774.823} C_VEL
LIN {X 0,Y 545.192,Z 176.574,A -85,B 0,C 180,E1 -3777.783,E2 -3777.783} C_VEL
LIN {X 0,Y 545.133,Z 176.655,A -85,B 0,C 180,E1 -3780.346,E2 -3780.346} C_VEL
LIN {X 0,Y 545.13,Z 193.473,A -85,B 0,C 180,E1 -3783.141,E2 -3783.141} C_VEL
LIN {X 0,Y 545.108,Z 207.57,A -85,B 0,C 180,E1 -3785.549,E2 -3785.549} C_VEL
LIN {X 0,Y 545.031,Z 223.454,A -85,B 0,C 180,E1 -3788.434,E2 -3788.434} C_VEL
LIN {X 0,Y 545.054,Z 224.4,A -85,B 0,C 180,E1 -3788.55,E2 -3788.55} C_VEL
LIN {X 0,Y 545.867,Z 230.743,A -85,B 0,C 180,E1 -3788.677,E2 -3788.677} C_VEL
LIN {X 0,Y 545.686,Z 300.962,A -85,B 0,C 180,E1 -3789.638,E2 -3789.638} C_VEL
LIN {X 0,Y 545.623,Z 311.588,A -85,B 0,C 180,E1 -3789.897,E2 -3789.897} C_VEL
LIN {X 0,Y 545.5,Z 323.366,A -85,B 0,C 180,E1 -3790.344,E2 -3790.344} C_VEL
LIN {X 0,Y 545.347,Z 333.144,A -85,B 0,C 180,E1 -3790.863,E2 -3790.863} C_VEL
LIN {X 0,Y 545.202,Z 342.337,A -85,B 0,C 180,E1 -3791.493,E2 -3791.493} C_VEL
LIN {X 0,Y 545.072,Z 350.464,A -85,B 0,C 180,E1 -3792.188,E2 -3792.188} C_VEL
LIN {X 0,Y 544.942,Z 358.499,A -85,B 0,C 180,E1 -3793.043,E2 -3793.043} C_VEL
LIN {X 0,Y 544.837,Z 365.521,A -85,B 0,C 180,E1 -3793.996,E2 -3793.996} C_VEL
LIN {X 0,Y 544.771,Z 371.081,A -85,B 0,C 180,E1 -3794.952,E2 -3794.952} C_VEL
LIN {X 0,Y 544.707,Z 374.698,A -85,B 0,C 180,E1 -3795.72,E2 -3795.72} C_VEL
LIN {X 0,Y 544.659,Z 378.825,A -85,B 0,C 180,E1 -3796.877,E2 -3796.877} C_VEL
LIN {X 0,Y 544.588,Z 381.646,A -85,B 0,C 180,E1 -3798.042,E2 -3798.042} C_VEL
LIN {X 0,Y 544.579,Z 382.742,A -85,B 0,C 180,E1 -3798.822,E2 -3798.822} C_VEL
LIN {X 0,Y 544.596,Z 383.299,A -85,B 0,C 180,E1 -3799.604,E2 -3799.604} C_VEL
LIN {X 0,Y 544.564,Z 383.338,A -85,B 0,C 180,E1 -3800.392,E2 -3800.392} C_VEL
LIN {X 0,Y 544.589,Z 382.385,A -85,B 0,C 180,E1 -3801.535,E2 -3801.535} C_VEL
LIN {X 0,Y 544.587,Z 381.76,A -85,B 0,C 180,E1 -3801.978,E2 -3801.978} C_VEL
LIN {X 0,Y 544.629,Z 378.903,A -85,B 0,C 180,E1 -3803.177,E2 -3803.177} C_VEL
LIN {X 0,Y 544.687,Z 376.225,A -85,B 0,C 180,E1 -3803.98,E2 -3803.98} C_VEL
LIN {X 0,Y 544.71,Z 373.579,A -85,B 0,C 180,E1 -3804.613,E2 -3804.613} C_VEL
LIN {X 0,Y 544.09,Z 371.014,A -85,B 0,C 180,E1 -3805.17,E2 -3805.17} C_VEL
LIN {X 0,Y 541.339,Z 366.39,A -85,B 0,C 180,E1 -3806.052,E2 -3806.052} C_VEL
LIN {X 0,Y 538.582,Z 360.943,A -85,B 0,C 180,E1 -3806.882,E2 -3806.882} C_VEL
LIN {X 0,Y 537.952,Z 357.086,A -85,B 0,C 180,E1 -3807.355,E2 -3807.355} C_VEL
LIN {X 0,Y 538.062,Z 349.307,A -85,B 0,C 180,E1 -3808.154,E2 -3808.154} C_VEL
LIN {X 0,Y 538.255,Z 340.405,A -85,B 0,C 180,E1 -3808.888,E2 -3808.888} C_VEL
LIN {X 0,Y 538.428,Z 329.884,A -85,B 0,C 180,E1 -3809.56,E2 -3809.56} C_VEL
LIN {X 0,Y 538.578,Z 319.567,A -85,B 0,C 180,E1 -3810.05,E2 -3810.05} C_VEL
LIN {X 0,Y 538.663,Z 308.507,A -85,B 0,C 180,E1 -3810.423,E2 -3810.423} C_VEL
LIN {X 0,Y 538.732,Z 296.901,A -85,B 0,C 180,E1 -3810.663,E2 -3810.663} C_VEL
LIN {X 0,Y 538.869,Z 230.021,A -85,B 0,C 180,E1 -3811.574,E2 -3811.574} C_VEL
LIN {X 0,Y 538.032,Z 224.515,A -85,B 0,C 180,E1 -3811.694,E2 -3811.694} C_VEL
LIN {X 0,Y 538.009,Z 221.969,A -85,B 0,C 180,E1 -3812.097,E2 -3812.097} C_VEL
LIN {X 0,Y 538.103,Z 209.887,A -85,B 0,C 180,E1 -3814.402,E2 -3814.402} C_VEL
LIN {X 0,Y 538.256,Z 196.464,A -85,B 0,C 180,E1 -3816.914,E2 -3816.914} C_VEL
LIN {X 0,Y 538.421,Z 181.433,A -85,B 0,C 180,E1 -3819.761,E2 -3819.761} C_VEL
LIN {X 0,Y 538.113,Z 177.486,A -85,B 0,C 180,E1 -3820.568,E2 -3820.568} C_VEL
LIN {X 0,Y 538.018,Z 177.469,A -85,B 0,C 180,E1 -3824.073,E2 -3824.073} C_VEL
LIN {X 0,Y 538.018,Z 177.465,A -85,B 0,C 180,E1 -3827.214,E2 -3827.214} C_VEL
LIN {X 0,Y 538.021,Z 177.464,A -85,B 0,C 180,E1 -3830.203,E2 -3830.203} C_VEL
LIN {X 0,Y 538.026,Z 177.462,A -85,B 0,C 180,E1 -3833.067,E2 -3833.067} C_VEL
LIN {X 0,Y 538.022,Z 177.467,A -85,B 0,C 180,E1 -3835.827,E2 -3835.827} C_VEL
LIN {X 0,Y 538.007,Z 177.463,A -85,B 0,C 180,E1 -3838.498,E2 -3838.498} C_VEL
LIN {X 0,Y 538.059,Z 177.46,A -85,B 0,C 180,E1 -3841.1,E2 -3841.1} C_VEL
LIN {X 0,Y 538.049,Z 177.465,A -85,B 0,C 180,E1 -3843.633,E2 -3843.633} C_VEL
LIN {X 0,Y 538.005,Z 177.464,A -85,B 0,C 180,E1 -3846.122,E2 -3846.122} C_VEL
LIN {X 0,Y 538.036,Z 177.468,A -85,B 0,C 180,E1 -3849.348,E2 -3849.348} C_VEL
LIN {X 0,Y 538.053,Z 177.458,A -85,B 0,C 180,E1 -3852.517,E2 -3852.517} C_VEL
LIN {X 0,Y 538.062,Z 177.461,A -85,B 0,C 180,E1 -3855.63,E2 -3855.63} C_VEL
LIN {X 0,Y 538.076,Z 177.456,A -85,B 0,C 180,E1 -3858.701,E2 -3858.701} C_VEL
LIN {X 0,Y 538.085,Z 177.455,A -85,B 0,C 180,E1 -3861.739,E2 -3861.739} C_VEL
LIN {X 0,Y 538.163,Z 177.447,A -85,B 0,C 180,E1 -3864.755,E2 -3864.755} C_VEL
LIN {X 0,Y 538.168,Z 177.444,A -85,B 0,C 180,E1 -3867.754,E2 -3867.754} C_VEL
LIN {X 0,Y 538.18,Z 177.446,A -85,B 0,C 180,E1 -3870.748,E2 -3870.748} C_VEL
LIN {X 0,Y 538.136,Z 177.456,A -85,B 0,C 180,E1 -3872.994,E2 -3872.994} C_VEL
LIN {X 0,Y 538.119,Z 177.449,A -85,B 0,C 180,E1 -3875.997,E2 -3875.997} C_VEL
LIN {X 0,Y 538.066,Z 177.464,A -85,B 0,C 180,E1 -3879.017,E2 -3879.017} C_VEL
LIN {X 0,Y 538.08,Z 177.454,A -85,B 0,C 180,E1 -3882.062,E2 -3882.062} C_VEL
LIN {X 0,Y 538.042,Z 177.464,A -85,B 0,C 180,E1 -3885.143,E2 -3885.143} C_VEL
LIN {X 0,Y 538.028,Z 177.463,A -85,B 0,C 180,E1 -3888.27,E2 -3888.27} C_VEL
LIN {X 0,Y 538.035,Z 177.467,A -85,B 0,C 180,E1 -3890.651,E2 -3890.651} C_VEL
LIN {X 0,Y 538.019,Z 177.462,A -85,B 0,C 180,E1 -3893.887,E2 -3893.887} C_VEL
LIN {X 0,Y 538.045,Z 177.463,A -85,B 0,C 180,E1 -3896.366,E2 -3896.366} C_VEL
LIN {X 0,Y 538.026,Z 177.465,A -85,B 0,C 180,E1 -3898.933,E2 -3898.933} C_VEL
LIN {X 0,Y 538.022,Z 177.462,A -85,B 0,C 180,E1 -3901.89,E2 -3901.89} C_VEL
LIN {X 0,Y 538.028,Z 177.469,A -85,B 0,C 180,E1 -3904.621,E2 -3904.621} C_VEL
LIN {X 0,Y 538.003,Z 177.465,A -85,B 0,C 180,E1 -3907.17,E2 -3907.17} C_VEL
LIN {X 0,Y 538.047,Z 177.459,A -85,B 0,C 180,E1 -3909.794,E2 -3909.794} C_VEL
LIN {X 0,Y 538.016,Z 177.466,A -85,B 0,C 180,E1 -3912.785,E2 -3912.785} C_VEL
LIN {X 0,Y 538.024,Z 177.461,A -85,B 0,C 180,E1 -3915.14,E2 -3915.14} C_VEL
LIN {X 0,Y 538.033,Z 177.468,A -85,B 0,C 180,E1 -3918.228,E2 -3918.228} C_VEL
LIN {X 0,Y 538.051,Z 177.465,A -85,B 0,C 180,E1 -3920.411,E2 -3920.411} C_VEL
LIN {X 0,Y 538.021,Z 177.462,A -85,B 0,C 180,E1 -3923.067,E2 -3923.067} C_VEL
LIN {X 0,Y 538.024,Z 177.465,A -85,B 0,C 180,E1 -3925.828,E2 -3925.828} C_VEL
LIN {X 0,Y 538.016,Z 177.466,A -85,B 0,C 180,E1 -3928.5,E2 -3928.5} C_VEL
LIN {X 0,Y 538.051,Z 177.458,A -85,B 0,C 180,E1 -3931.1,E2 -3931.1} C_VEL
LIN {X 0,Y 538.034,Z 177.463,A -85,B 0,C 180,E1 -3933.633,E2 -3933.633} C_VEL
LIN {X 0,Y 538.014,Z 177.471,A -85,B 0,C 180,E1 -3936.118,E2 -3936.118} C_VEL
LIN {X 0,Y 538.034,Z 177.461,A -85,B 0,C 180,E1 -3939.349,E2 -3939.349} C_VEL
LIN {X 0,Y 538.064,Z 177.458,A -85,B 0,C 180,E1 -3942.518,E2 -3942.518} C_VEL
LIN {X 0,Y 538.055,Z 177.462,A -85,B 0,C 180,E1 -3945.631,E2 -3945.631} C_VEL
LIN {X 0,Y 538.081,Z 177.454,A -85,B 0,C 180,E1 -3948.702,E2 -3948.702} C_VEL
LIN {X 0,Y 538.078,Z 177.463,A -85,B 0,C 180,E1 -3951.74,E2 -3951.74} C_VEL
LIN {X 0,Y 538.154,Z 177.445,A -85,B 0,C 180,E1 -3954.755,E2 -3954.755} C_VEL
LIN {X 0,Y 538.157,Z 177.453,A -85,B 0,C 180,E1 -3957.755,E2 -3957.755} C_VEL
LIN {X 0,Y 538.175,Z 177.442,A -85,B 0,C 180,E1 -3960.749,E2 -3960.749} C_VEL
LIN {X 0,Y 538.131,Z 177.449,A -85,B 0,C 180,E1 -3962.995,E2 -3962.995} C_VEL
LIN {X 0,Y 538.112,Z 177.453,A -85,B 0,C 180,E1 -3965.998,E2 -3965.998} C_VEL
LIN {X 0,Y 538.053,Z 177.46,A -85,B 0,C 180,E1 -3969.018,E2 -3969.018} C_VEL
LIN {X 0,Y 538.075,Z 177.456,A -85,B 0,C 180,E1 -3972.063,E2 -3972.063} C_VEL
LIN {X 0,Y 538.037,Z 177.464,A -85,B 0,C 180,E1 -3975.144,E2 -3975.144} C_VEL
LIN {X 0,Y 538.02,Z 177.462,A -85,B 0,C 180,E1 -3978.271,E2 -3978.271} C_VEL
LIN {X 0,Y 538.03,Z 177.461,A -85,B 0,C 180,E1 -3980.652,E2 -3980.652} C_VEL
LIN {X 0,Y 537.996,Z 177.466,A -85,B 0,C 180,E1 -3983.889,E2 -3983.889} C_VEL
LIN {X 0,Y 538.034,Z 177.46,A -85,B 0,C 180,E1 -3986.367,E2 -3986.367} C_VEL
LIN {X 0,Y 538.023,Z 177.466,A -85,B 0,C 180,E1 -3988.934,E2 -3988.934} C_VEL
LIN {X 0,Y 538.004,Z 177.464,A -85,B 0,C 180,E1 -3991.888,E2 -3991.888} C_VEL
LIN {X 0,Y 538.004,Z 177.466,A -85,B 0,C 180,E1 -3994.618,E2 -3994.618} C_VEL
LIN {X 0,Y 537.998,Z 177.473,A -85,B 0,C 180,E1 -3997.171,E2 -3997.171} C_VEL
LIN {X 0,Y 538.016,Z 177.463,A -85,B 0,C 180,E1 -3999.798,E2 -3999.798} C_VEL
LIN {X 0,Y 538.014,Z 177.468,A -85,B 0,C 180,E1 -4002.787,E2 -4002.787} C_VEL
LIN {X 0,Y 538.015,Z 177.462,A -85,B 0,C 180,E1 -4005.928,E2 -4005.928} C_VEL
LIN {X 0,Y 538.019,Z 177.466,A -85,B 0,C 180,E1 -4009.257,E2 -4009.257} C_VEL
LIN {X 0,Y 537.986,Z 177.466,A -85,B 0,C 180,E1 -4012.123,E2 -4012.123} C_VEL
LIN {X 0,Y 537.992,Z 177.474,A -85,B 0,C 180,E1 -4014.916,E2 -4014.916} C_VEL
LIN {X 0,Y 538.015,Z 177.464,A -85,B 0,C 180,E1 -4017.618,E2 -4017.618} C_VEL
LIN {X 0,Y 538.005,Z 177.468,A -85,B 0,C 180,E1 -4020.239,E2 -4020.239} C_VEL
LIN {X 0,Y 538.032,Z 177.468,A -85,B 0,C 180,E1 -4022.795,E2 -4022.795} C_VEL
LIN {X 0,Y 538.045,Z 177.694,A -85,B 0,C 180,E1 -4024.7,E2 -4024.7} C_VEL
LIN {X 0,Y 539.992,Z 186.526,A -85,B 0,C 180,E1 -4025.864,E2 -4025.864} C_VEL
LIN {X 0,Y 539.714,Z 203.098,A -85,B 0,C 180,E1 -4027.814,E2 -4027.814} C_VEL
LIN {X 0,Y 539.205,Z 226.971,A -85,B 0,C 180,E1 -4030.588,E2 -4030.588} C_VEL
LIN {X 0,Y 538.769,Z 252.541,A -85,B 0,C 180,E1 -4033.518,E2 -4033.518} C_VEL
LIN {X 0,Y 538.567,Z 268.084,A -85,B 0,C 180,E1 -4035.264,E2 -4035.264} C_VEL
LIN {X 0,Y 539.548,Z 277.564,A -85,B 0,C 180,E1 -4035.44,E2 -4035.44} C_VEL
LIN {X 0,Y 539.224,Z 377.832,A -85,B 0,C 180,E1 -4036.792,E2 -4036.792} C_VEL
LIN {X 0,Y 539.039,Z 391.213,A -85,B 0,C 180,E1 -4037.123,E2 -4037.123} C_VEL
LIN {X 0,Y 538.852,Z 403.464,A -85,B 0,C 180,E1 -4037.573,E2 -4037.573} C_VEL
LIN {X 0,Y 538.653,Z 415.763,A -85,B 0,C 180,E1 -4038.187,E2 -4038.187} C_VEL
LIN {X 0,Y 538.465,Z 426.842,A -85,B 0,C 180,E1 -4038.901,E2 -4038.901} C_VEL
LIN {X 0,Y 538.199,Z 437.467,A -85,B 0,C 180,E1 -4039.752,E2 -4039.752} C_VEL
LIN {X 0,Y 538.026,Z 446.156,A -85,B 0,C 180,E1 -4040.603,E2 -4040.603} C_VEL
LIN {X 0,Y 537.913,Z 454.171,A -85,B 0,C 180,E1 -4041.548,E2 -4041.548} C_VEL
LIN {X 0,Y 537.754,Z 461.993,A -85,B 0,C 180,E1 -4042.68,E2 -4042.68} C_VEL
LIN {X 0,Y 537.674,Z 469.196,A -85,B 0,C 180,E1 -4043.998,E2 -4043.998} C_VEL
LIN {X 0,Y 537.54,Z 473.98,A -85,B 0,C 180,E1 -4045.126,E2 -4045.126} C_VEL
LIN {X 0,Y 537.591,Z 477.649,A -85,B 0,C 180,E1 -4046.253,E2 -4046.253} C_VEL
LIN {X 0,Y 537.58,Z 479.537,A -85,B 0,C 180,E1 -4047.003,E2 -4047.003} C_VEL
LIN {X 0,Y 537.451,Z 481.953,A -85,B 0,C 180,E1 -4048.502,E2 -4048.502} C_VEL
LIN {X 0,Y 537.445,Z 482.569,A -85,B 0,C 180,E1 -4049.251,E2 -4049.251} C_VEL
LIN {X 0,Y 537.445,Z 482.787,A -85,B 0,C 180,E1 -4050.001,E2 -4050.001} C_VEL
LIN {X 0,Y 537.445,Z 482.568,A -85,B 0,C 180,E1 -4050.75,E2 -4050.75} C_VEL
LIN {X 0,Y 537.49,Z 480.944,A -85,B 0,C 180,E1 -4052.249,E2 -4052.249} C_VEL
LIN {X 0,Y 537.58,Z 479.533,A -85,B 0,C 180,E1 -4052.998,E2 -4052.998} C_VEL
LIN {X 0,Y 537.604,Z 476.552,A -85,B 0,C 180,E1 -4054.124,E2 -4054.124} C_VEL
LIN {X 0,Y 537.588,Z 472.509,A -85,B 0,C 180,E1 -4055.251,E2 -4055.251} C_VEL
LIN {X 0,Y 537.658,Z 466.297,A -85,B 0,C 180,E1 -4056.567,E2 -4056.567} C_VEL
LIN {X 0,Y 537.798,Z 459.504,A -85,B 0,C 180,E1 -4057.698,E2 -4057.698} C_VEL
LIN {X 0,Y 537.949,Z 451.072,A -85,B 0,C 180,E1 -4058.831,E2 -4058.831} C_VEL
LIN {X 0,Y 538.082,Z 442.403,A -85,B 0,C 180,E1 -4059.776,E2 -4059.776} C_VEL
LIN {X 0,Y 538.33,Z 431.703,A -85,B 0,C 180,E1 -4060.722,E2 -4060.722} C_VEL
LIN {X 0,Y 538.525,Z 420.279,A -85,B 0,C 180,E1 -4061.533,E2 -4061.533} C_VEL
LIN {X 0,Y 538.782,Z 408.382,A -85,B 0,C 180,E1 -4062.19,E2 -4062.19} C_VEL
LIN {X 0,Y 538.971,Z 395.889,A -85,B 0,C 180,E1 -4062.712,E2 -4062.712} C_VEL
LIN {X 0,Y 539.149,Z 383.029,A -85,B 0,C 180,E1 -4063.091,E2 -4063.091} C_VEL
LIN {X 0,Y 539.238,Z 369.418,A -85,B 0,C 180,E1 -4063.328,E2 -4063.328} C_VEL
LIN {X 0,Y 539.383,Z 275.38,A -85,B 0,C 180,E1 -4064.587,E2 -4064.587} C_VEL
LIN {X 0,Y 538.548,Z 267.781,A -85,B 0,C 180,E1 -4064.737,E2 -4064.737} C_VEL
LIN {X 0,Y 538.9,Z 240.053,A -85,B 0,C 180,E1 -4067.819,E2 -4067.819} C_VEL
LIN {X 0,Y 539.306,Z 211.968,A -85,B 0,C 180,E1 -4071,E2 -4071} C_VEL
LIN {X 0,Y 539.697,Z 186.153,A -85,B 0,C 180,E1 -4073.928,E2 -4073.928} C_VEL
LIN {X 0,Y 538.076,Z 177.599,A -85,B 0,C 180,E1 -4075.003,E2 -4075.003} C_VEL
LIN {X 0,Y 537.999,Z 177.468,A -85,B 0,C 180,E1 -4078.052,E2 -4078.052} C_VEL
LIN {X 0,Y 538.01,Z 177.467,A -85,B 0,C 180,E1 -4080.628,E2 -4080.628} C_VEL
LIN {X 0,Y 538.023,Z 177.47,A -85,B 0,C 180,E1 -4083.278,E2 -4083.278} C_VEL
LIN {X 0,Y 537.992,Z 177.467,A -85,B 0,C 180,E1 -4086.005,E2 -4086.005} C_VEL
LIN {X 0,Y 538.012,Z 177.469,A -85,B 0,C 180,E1 -4088.831,E2 -4088.831} C_VEL
LIN {X 0,Y 538,Z 177.466,A -85,B 0,C 180,E1 -4091.875,E2 -4091.875} C_VEL
LIN {X 0,Y 538.003,Z 177.471,A -85,B 0,C 180,E1 -4094.863,E2 -4094.863} C_VEL
LIN {X 0,Y 537.99,Z 177.471,A -85,B 0,C 180,E1 -4097.211,E2 -4097.211} C_VEL
LIN {X 0,Y 538.023,Z 177.462,A -85,B 0,C 180,E1 -4100.203,E2 -4100.203} C_VEL
LIN {X 0,Y 538.026,Z 177.468,A -85,B 0,C 180,E1 -4103.067,E2 -4103.067} C_VEL
LIN {X 0,Y 538.012,Z 177.463,A -85,B 0,C 180,E1 -4105.826,E2 -4105.826} C_VEL
LIN {X 0,Y 538.01,Z 177.469,A -85,B 0,C 180,E1 -4108.498,E2 -4108.498} C_VEL
LIN {X 0,Y 538.021,Z 177.466,A -85,B 0,C 180,E1 -4111.097,E2 -4111.097} C_VEL
LIN {X 0,Y 538.04,Z 177.46,A -85,B 0,C 180,E1 -4113.633,E2 -4113.633} C_VEL
LIN {X 0,Y 538.009,Z 177.466,A -85,B 0,C 180,E1 -4116.122,E2 -4116.122} C_VEL
LIN {X 0,Y 538.038,Z 177.461,A -85,B 0,C 180,E1 -4119.348,E2 -4119.348} C_VEL
LIN {X 0,Y 538.037,Z 177.469,A -85,B 0,C 180,E1 -4122.467,E2 -4122.467} C_VEL
LIN {X 0,Y 538.063,Z 177.458,A -85,B 0,C 180,E1 -4125.63,E2 -4125.63} C_VEL
LIN {X 0,Y 538.078,Z 177.461,A -85,B 0,C 180,E1 -4128.701,E2 -4128.701} C_VEL
LIN {X 0,Y 538.063,Z 177.459,A -85,B 0,C 180,E1 -4131.739,E2 -4131.739} C_VEL
LIN {X 0,Y 538.156,Z 177.45,A -85,B 0,C 180,E1 -4134.755,E2 -4134.755} C_VEL
LIN {X 0,Y 538.164,Z 177.449,A -85,B 0,C 180,E1 -4137.754,E2 -4137.754} C_VEL
LIN {X 0,Y 538.111,Z 177.557,A -85,B 0,C 180,E1 -4140.35,E2 -4140.35} C_VEL
LIN {X 0,Y 538.058,Z 193.484,A -85,B 0,C 180,E1 -4142.995,E2 -4142.995} C_VEL
LIN {X 0,Y 538.036,Z 209.966,A -85,B 0,C 180,E1 -4145.81,E2 -4145.81} C_VEL
LIN {X 0,Y 538.027,Z 224.372,A -85,B 0,C 180,E1 -4148.355,E2 -4148.355} C_VEL
LIN {X 0,Y 538.83,Z 229.696,A -85,B 0,C 180,E1 -4148.485,E2 -4148.485} C_VEL
LIN {X 0,Y 538.742,Z 301.928,A -85,B 0,C 180,E1 -4149.503,E2 -4149.503} C_VEL
LIN {X 0,Y 538.617,Z 313.88,A -85,B 0,C 180,E1 -4149.813,E2 -4149.813} C_VEL
LIN {X 0,Y 538.495,Z 324.557,A -85,B 0,C 180,E1 -4150.243,E2 -4150.243} C_VEL
LIN {X 0,Y 538.359,Z 334.956,A -85,B 0,C 180,E1 -4150.816,E2 -4150.816} C_VEL
LIN {X 0,Y 538.209,Z 344.289,A -85,B 0,C 180,E1 -4151.482,E2 -4151.482} C_VEL
LIN {X 0,Y 538.066,Z 352.846,A -85,B 0,C 180,E1 -4152.254,E2 -4152.254} C_VEL
LIN {X 0,Y 537.872,Z 361.229,A -85,B 0,C 180,E1 -4153.218,E2 -4153.218} C_VEL
LIN {X 0,Y 537.826,Z 367.819,A -85,B 0,C 180,E1 -4154.182,E2 -4154.182} C_VEL
LIN {X 0,Y 537.712,Z 373.097,A -85,B 0,C 180,E1 -4155.153,E2 -4155.153} C_VEL
LIN {X 0,Y 537.639,Z 377.904,A -85,B 0,C 180,E1 -4156.322,E2 -4156.322} C_VEL
LIN {X 0,Y 537.559,Z 381.227,A -85,B 0,C 180,E1 -4157.499,E2 -4157.499} C_VEL
LIN {X 0,Y 537.52,Z 382.749,A -85,B 0,C 180,E1 -4158.288,E2 -4158.288} C_VEL
LIN {X 0,Y 537.531,Z 383.702,A -85,B 0,C 180,E1 -4159.078,E2 -4159.078} C_VEL
LIN {X 0,Y 537.528,Z 384.074,A -85,B 0,C 180,E1 -4159.873,E2 -4159.873} C_VEL
LIN {X 0,Y 537.495,Z 383.888,A -85,B 0,C 180,E1 -4160.673,E2 -4160.673} C_VEL
LIN {X 0,Y 537.552,Z 382.662,A -85,B 0,C 180,E1 -4161.835,E2 -4161.835} C_VEL
LIN {X 0,Y 537.56,Z 379.918,A -85,B 0,C 180,E1 -4163.092,E2 -4163.092} C_VEL
LIN {X 0,Y 537.641,Z 377.333,A -85,B 0,C 180,E1 -4163.905,E2 -4163.905} C_VEL
LIN {X 0,Y 537.695,Z 373.017,A -85,B 0,C 180,E1 -4164.931,E2 -4164.931} C_VEL
LIN {X 0,Y 537.764,Z 367.6,A -85,B 0,C 180,E1 -4165.922,E2 -4165.922} C_VEL
LIN {X 0,Y 537.862,Z 361.642,A -85,B 0,C 180,E1 -4166.794,E2 -4166.794} C_VEL
LIN {X 0,Y 537.952,Z 357.086,A -85,B 0,C 180,E1 -4167.355,E2 -4167.355} C_VEL
LIN {X 0,Y 537.332,Z 353.094,A -85,B 0,C 180,E1 -4167.807,E2 -4167.807} C_VEL
LIN {X 0,Y 534.627,Z 346.23,A -85,B 0,C 180,E1 -4168.511,E2 -4168.511} C_VEL
LIN {X 0,Y 531.972,Z 338.722,A -85,B 0,C 180,E1 -4169.152,E2 -4169.152} C_VEL
LIN {X 0,Y 531.421,Z 333.706,A -85,B 0,C 180,E1 -4169.491,E2 -4169.491} C_VEL
LIN {X 0,Y 531.552,Z 323.231,A -85,B 0,C 180,E1 -4170.05,E2 -4170.05} C_VEL
LIN {X 0,Y 531.684,Z 311.233,A -85,B 0,C 180,E1 -4170.5,E2 -4170.5} C_VEL
LIN {X 0,Y 531.747,Z 300.682,A -85,B 0,C 180,E1 -4170.752,E2 -4170.752} C_VEL
LIN {X 0,Y 531.95,Z 230.881,A -85,B 0,C 180,E1 -4171.732,E2 -4171.732} C_VEL
LIN {X 0,Y 531.03,Z 224.816,A -85,B 0,C 180,E1 -4171.861,E2 -4171.861} C_VEL
LIN {X 0,Y 530.973,Z 223.085,A -85,B 0,C 180,E1 -4172.101,E2 -4172.101} C_VEL
LIN {X 0,Y 531.121,Z 208.506,A -85,B 0,C 180,E1 -4174.874,E2 -4174.874} C_VEL
LIN {X 0,Y 531.292,Z 194.724,A -85,B 0,C 180,E1 -4177.48,E2 -4177.48} C_VEL
LIN {X 0,Y 531.376,Z 180.799,A -85,B 0,C 180,E1 -4180.118,E2 -4180.118} C_VEL
LIN {X 0,Y 531.06,Z 178.364,A -85,B 0,C 180,E1 -4180.648,E2 -4180.648} C_VEL
LIN {X 0,Y 530.953,Z 178.348,A -85,B 0,C 180,E1 -4183.495,E2 -4183.495} C_VEL
LIN {X 0,Y 530.953,Z 178.344,A -85,B 0,C 180,E1 -4186.504,E2 -4186.504} C_VEL
LIN {X 0,Y 530.984,Z 178.339,A -85,B 0,C 180,E1 -4188.976,E2 -4188.976} C_VEL
LIN {X 0,Y 530.955,Z 178.349,A -85,B 0,C 180,E1 -4191.529,E2 -4191.529} C_VEL
LIN {X 0,Y 530.975,Z 178.34,A -85,B 0,C 180,E1 -4194.381,E2 -4194.381} C_VEL
LIN {X 0,Y 530.965,Z 178.343,A -85,B 0,C 180,E1 -4197.133,E2 -4197.133} C_VEL
LIN {X 0,Y 530.968,Z 178.345,A -85,B 0,C 180,E1 -4199.803,E2 -4199.803} C_VEL
LIN {X 0,Y 531.015,Z 178.334,A -85,B 0,C 180,E1 -4202.466,E2 -4202.466} C_VEL
LIN {X 0,Y 531.007,Z 178.337,A -85,B 0,C 180,E1 -4204.942,E2 -4204.942} C_VEL
LIN {X 0,Y 530.97,Z 178.34,A -85,B 0,C 180,E1 -4208.246,E2 -4208.246} C_VEL
LIN {X 0,Y 530.991,Z 178.338,A -85,B 0,C 180,E1 -4210.677,E2 -4210.677} C_VEL
LIN {X 0,Y 530.985,Z 178.343,A -85,B 0,C 180,E1 -4213.071,E2 -4213.071} C_VEL
LIN {X 0,Y 531.039,Z 178.338,A -85,B 0,C 180,E1 -4215.436,E2 -4215.436} C_VEL
LIN {X 0,Y 531.036,Z 178.332,A -85,B 0,C 180,E1 -4218.549,E2 -4218.549} C_VEL
LIN {X 0,Y 531.055,Z 178.332,A -85,B 0,C 180,E1 -4221.629,E2 -4221.629} C_VEL
LIN {X 0,Y 531.122,Z 178.323,A -85,B 0,C 180,E1 -4224.685,E2 -4224.685} C_VEL
LIN {X 0,Y 531.14,Z 178.32,A -85,B 0,C 180,E1 -4227.724,E2 -4227.724} C_VEL
LIN {X 0,Y 531.15,Z 178.322,A -85,B 0,C 180,E1 -4230.758,E2 -4230.758} C_VEL
LIN {X 0,Y 531.103,Z 178.333,A -85,B 0,C 180,E1 -4233.034,E2 -4233.034} C_VEL
LIN {X 0,Y 531.074,Z 178.327,A -85,B 0,C 180,E1 -4236.077,E2 -4236.077} C_VEL
LIN {X 0,Y 531.052,Z 178.331,A -85,B 0,C 180,E1 -4238.37,E2 -4238.37} C_VEL
LIN {X 0,Y 531.048,Z 178.33,A -85,B 0,C 180,E1 -4241.672,E2 -4241.672} C_VEL
LIN {X 0,Y 531.027,Z 178.34,A -85,B 0,C 180,E1 -4244.955,E2 -4244.955} C_VEL
LIN {X 0,Y 531.012,Z 178.334,A -85,B 0,C 180,E1 -4247.722,E2 -4247.722} C_VEL
LIN {X 0,Y 530.995,Z 178.343,A -85,B 0,C 180,E1 -4250.937,E2 -4250.937} C_VEL
LIN {X 0,Y 530.975,Z 178.342,A -85,B 0,C 180,E1 -4254.224,E2 -4254.224} C_VEL
LIN {X 0,Y 531.007,Z 178.343,A -85,B 0,C 180,E1 -4256.743,E2 -4256.743} C_VEL
LIN {X 0,Y 530.977,Z 178.34,A -85,B 0,C 180,E1 -4259.322,E2 -4259.322} C_VEL
LIN {X 0,Y 530.974,Z 178.342,A -85,B 0,C 180,E1 -4262.102,E2 -4262.102} C_VEL
LIN {X 0,Y 530.985,Z 178.342,A -85,B 0,C 180,E1 -4264.854,E2 -4264.854} C_VEL
LIN {X 0,Y 530.96,Z 178.341,A -85,B 0,C 180,E1 -4267.507,E2 -4267.507} C_VEL
LIN {X 0,Y 531.019,Z 178.343,A -85,B 0,C 180,E1 -4270.428,E2 -4270.428} C_VEL
LIN {X 0,Y 530.958,Z 178.341,A -85,B 0,C 180,E1 -4273.494,E2 -4273.494} C_VEL
LIN {X 0,Y 530.951,Z 178.349,A -85,B 0,C 180,E1 -4276.505,E2 -4276.505} C_VEL
LIN {X 0,Y 531,Z 178.337,A -85,B 0,C 180,E1 -4279.569,E2 -4279.569} C_VEL
LIN {X 0,Y 530.961,Z 178.345,A -85,B 0,C 180,E1 -4282.576,E2 -4282.576} C_VEL
LIN {X 0,Y 530.995,Z 178.337,A -85,B 0,C 180,E1 -4285.311,E2 -4285.311} C_VEL
LIN {X 0,Y 530.975,Z 178.346,A -85,B 0,C 180,E1 -4288.033,E2 -4288.033} C_VEL
LIN {X 0,Y 530.999,Z 178.337,A -85,B 0,C 180,E1 -4290.87,E2 -4290.87} C_VEL
LIN {X 0,Y 530.997,Z 178.337,A -85,B 0,C 180,E1 -4293.256,E2 -4293.256} C_VEL
LIN {X 0,Y 530.988,Z 178.345,A -85,B 0,C 180,E1 -4295.958,E2 -4295.958} C_VEL
LIN {X 0,Y 530.993,Z 178.337,A -85,B 0,C 180,E1 -4299.062,E2 -4299.062} C_VEL
LIN {X 0,Y 531.008,Z 178.339,A -85,B 0,C 180,E1 -4302.278,E2 -4302.278} C_VEL
LIN {X 0,Y 531.01,Z 178.337,A -85,B 0,C 180,E1 -4305.436,E2 -4305.436} C_VEL
LIN {X 0,Y 531.038,Z 178.332,A -85,B 0,C 180,E1 -4308.55,E2 -4308.55} C_VEL
LIN {X 0,Y 531.048,Z 178.337,A -85,B 0,C 180,E1 -4311.63,E2 -4311.63} C_VEL
LIN {X 0,Y 531.113,Z 178.322,A -85,B 0,C 180,E1 -4314.686,E2 -4314.686} C_VEL
LIN {X 0,Y 531.129,Z 178.329,A -85,B 0,C 180,E1 -4317.725,E2 -4317.725} C_VEL
LIN {X 0,Y 531.145,Z 178.318,A -85,B 0,C 180,E1 -4320.759,E2 -4320.759} C_VEL
LIN {X 0,Y 531.098,Z 178.325,A -85,B 0,C 180,E1 -4323.035,E2 -4323.035} C_VEL
LIN {X 0,Y 531.068,Z 178.33,A -85,B 0,C 180,E1 -4326.078,E2 -4326.078} C_VEL
LIN {X 0,Y 531.042,Z 178.331,A -85,B 0,C 180,E1 -4328.371,E2 -4328.371} C_VEL
LIN {X 0,Y 531.043,Z 178.337,A -85,B 0,C 180,E1 -4331.672,E2 -4331.672} C_VEL
LIN {X 0,Y 531.023,Z 178.336,A -85,B 0,C 180,E1 -4334.956,E2 -4334.956} C_VEL
LIN {X 0,Y 531.009,Z 178.339,A -85,B 0,C 180,E1 -4337.723,E2 -4337.723} C_VEL
LIN {X 0,Y 531.017,Z 178.334,A -85,B 0,C 180,E1 -4340.128,E2 -4340.128} C_VEL
LIN {X 0,Y 530.938,Z 178.344,A -85,B 0,C 180,E1 -4342.574,E2 -4342.574} C_VEL
LIN {X 0,Y 530.987,Z 178.343,A -85,B 0,C 180,E1 -4345.059,E2 -4345.059} C_VEL
LIN {X 0,Y 531.004,Z 178.339,A -85,B 0,C 180,E1 -4347.596,E2 -4347.596} C_VEL
LIN {X 0,Y 530.968,Z 178.342,A -85,B 0,C 180,E1 -4350.646,E2 -4350.646} C_VEL
LIN {X 0,Y 530.95,Z 178.344,A -85,B 0,C 180,E1 -4353.776,E2 -4353.776} C_VEL
LIN {X 0,Y 530.949,Z 178.344,A -85,B 0,C 180,E1 -4356.559,E2 -4356.559} C_VEL
LIN {X 0,Y 530.979,Z 178.342,A -85,B 0,C 180,E1 -4359.444,E2 -4359.444} C_VEL
LIN {X 0,Y 530.973,Z 178.341,A -85,B 0,C 180,E1 -4362.458,E2 -4362.458} C_VEL
LIN {X 0,Y 530.978,Z 178.34,A -85,B 0,C 180,E1 -4365.622,E2 -4365.622} C_VEL
LIN {X 0,Y 530.975,Z 178.343,A -85,B 0,C 180,E1 -4368.564,E2 -4368.564} C_VEL
LIN {X 0,Y 530.952,Z 178.343,A -85,B 0,C 180,E1 -4371.53,E2 -4371.53} C_VEL
LIN {X 0,Y 530.947,Z 178.345,A -85,B 0,C 180,E1 -4374.38,E2 -4374.38} C_VEL
LIN {X 0,Y 530.965,Z 178.346,A -85,B 0,C 180,E1 -4377.134,E2 -4377.134} C_VEL
LIN {X 0,Y 530.951,Z 178.345,A -85,B 0,C 180,E1 -4379.803,E2 -4379.803} C_VEL
LIN {X 0,Y 530.974,Z 178.348,A -85,B 0,C 180,E1 -4382.476,E2 -4382.476} C_VEL
LIN {X 0,Y 531.004,Z 178.517,A -85,B 0,C 180,E1 -4384.48,E2 -4384.48} C_VEL
LIN {X 0,Y 533.178,Z 189.03,A -85,B 0,C 180,E1 -4385.883,E2 -4385.883} C_VEL
LIN {X 0,Y 532.598,Z 212.908,A -85,B 0,C 180,E1 -4388.724,E2 -4388.724} C_VEL
LIN {X 0,Y 532.022,Z 239.486,A -85,B 0,C 180,E1 -4391.834,E2 -4391.834} C_VEL
LIN {X 0,Y 531.558,Z 265.488,A -85,B 0,C 180,E1 -4394.835,E2 -4394.835} C_VEL
LIN {X 0,Y 531.568,Z 268.139,A -85,B 0,C 180,E1 -4395.102,E2 -4395.102} C_VEL
LIN {X 0,Y 532.632,Z 278.162,A -85,B 0,C 180,E1 -4395.279,E2 -4395.279} C_VEL
LIN {X 0,Y 532.251,Z 377.394,A -85,B 0,C 180,E1 -4396.64,E2 -4396.64} C_VEL
LIN {X 0,Y 532.075,Z 390.757,A -85,B 0,C 180,E1 -4396.976,E2 -4396.976} C_VEL
LIN {X 0,Y 531.861,Z 403.558,A -85,B 0,C 180,E1 -4397.456,E2 -4397.456} C_VEL
LIN {X 0,Y 531.614,Z 416.294,A -85,B 0,C 180,E1 -4398.114,E2 -4398.114} C_VEL
LIN {X 0,Y 531.409,Z 427.319,A -85,B 0,C 180,E1 -4398.848,E2 -4398.848} C_VEL
LIN {X 0,Y 531.139,Z 437.764,A -85,B 0,C 180,E1 -4399.711,E2 -4399.711} C_VEL
LIN {X 0,Y 530.924,Z 447.139,A -85,B 0,C 180,E1 -4400.669,E2 -4400.669} C_VEL
LIN {X 0,Y 530.756,Z 456.242,A -85,B 0,C 180,E1 -4401.817,E2 -4401.817} C_VEL
LIN {X 0,Y 530.626,Z 463.571,A -85,B 0,C 180,E1 -4402.963,E2 -4402.963} C_VEL
LIN {X 0,Y 530.592,Z 470.253,A -85,B 0,C 180,E1 -4404.299,E2 -4404.299} C_VEL
LIN {X 0,Y 530.463,Z 474.657,A -85,B 0,C 180,E1 -4405.441,E2 -4405.441} C_VEL
LIN {X 0,Y 530.516,Z 476.997,A -85,B 0,C 180,E1 -4406.203,E2 -4406.203} C_VEL
LIN {X 0,Y 530.512,Z 478.889,A -85,B 0,C 180,E1 -4406.963,E2 -4406.963} C_VEL
LIN {X 0,Y 530.378,Z 481.309,A -85,B 0,C 180,E1 -4408.482,E2 -4408.482} C_VEL
LIN {X 0,Y 530.373,Z 481.925,A -85,B 0,C 180,E1 -4409.241,E2 -4409.241} C_VEL
LIN {X 0,Y 530.375,Z 482.141,A -85,B 0,C 180,E1 -4410.001,E2 -4410.001} C_VEL
LIN {X 0,Y 530.374,Z 481.918,A -85,B 0,C 180,E1 -4410.76,E2 -4410.76} C_VEL
LIN {X 0,Y 530.418,Z 480.285,A -85,B 0,C 180,E1 -4412.279,E2 -4412.279} C_VEL
LIN {X 0,Y 530.512,Z 478.864,A -85,B 0,C 180,E1 -4413.038,E2 -4413.038} C_VEL
LIN {X 0,Y 530.522,Z 475.868,A -85,B 0,C 180,E1 -4414.179,E2 -4414.179} C_VEL
LIN {X 0,Y 530.525,Z 471.809,A -85,B 0,C 180,E1 -4415.321,E2 -4415.321} C_VEL
LIN {X 0,Y 530.562,Z 466.154,A -85,B 0,C 180,E1 -4416.546,E2 -4416.546} C_VEL
LIN {X 0,Y 530.72,Z 458.748,A -85,B 0,C 180,E1 -4417.802,E2 -4417.802} C_VEL
LIN {X 0,Y 530.875,Z 450.278,A -85,B 0,C 180,E1 -4418.949,E2 -4418.949} C_VEL
LIN {X 0,Y 531.024,Z 441.557,A -85,B 0,C 180,E1 -4419.908,E2 -4419.908} C_VEL
LIN {X 0,Y 531.307,Z 430.809,A -85,B 0,C 180,E1 -4420.865,E2 -4420.865} C_VEL
LIN {X 0,Y 531.501,Z 419.934,A -85,B 0,C 180,E1 -4421.647,E2 -4421.647} C_VEL
LIN {X 0,Y 531.762,Z 408.279,A -85,B 0,C 180,E1 -4422.305,E2 -4422.305} C_VEL
LIN {X 0,Y 531.982,Z 395.936,A -85,B 0,C 180,E1 -4422.833,E2 -4422.833} C_VEL
LIN {X 0,Y 532.155,Z 383.333,A -85,B 0,C 180,E1 -4423.217,E2 -4423.217} C_VEL
LIN {X 0,Y 532.284,Z 370.514,A -85,B 0,C 180,E1 -4423.457,E2 -4423.457} C_VEL
LIN {X 0,Y 532.484,Z 276.149,A -85,B 0,C 180,E1 -4424.742,E2 -4424.742} C_VEL
LIN {X 0,Y 531.514,Z 267.411,A -85,B 0,C 180,E1 -4424.916,E2 -4424.916} C_VEL
LIN {X 0,Y 531.908,Z 240.456,A -85,B 0,C 180,E1 -4427.95,E2 -4427.95} C_VEL
LIN {X 0,Y 532.344,Z 213.003,A -85,B 0,C 180,E1 -4431.085,E2 -4431.085} C_VEL
LIN {X 0,Y 532.787,Z 188.269,A -85,B 0,C 180,E1 -4433.931,E2 -4433.931} C_VEL
LIN {X 0,Y 531.533,Z 180.87,A -85,B 0,C 180,E1 -4434.838,E2 -4434.838} C_VEL
LIN {X 0,Y 531.027,Z 178.447,A -85,B 0,C 180,E1 -4435.188,E2 -4435.188} C_VEL
LIN {X 0,Y 530.96,Z 178.345,A -85,B 0,C 180,E1 -4438.458,E2 -4438.458} C_VEL
LIN {X 0,Y 530.954,Z 178.351,A -85,B 0,C 180,E1 -4441.08,E2 -4441.08} C_VEL
LIN {X 0,Y 530.958,Z 178.345,A -85,B 0,C 180,E1 -4443.775,E2 -4443.775} C_VEL
LIN {X 0,Y 530.953,Z 178.346,A -85,B 0,C 180,E1 -4446.559,E2 -4446.559} C_VEL
LIN {X 0,Y 530.972,Z 178.345,A -85,B 0,C 180,E1 -4449.445,E2 -4449.445} C_VEL
LIN {X 0,Y 530.94,Z 178.347,A -85,B 0,C 180,E1 -4452.461,E2 -4452.461} C_VEL
LIN {X 0,Y 530.97,Z 178.343,A -85,B 0,C 180,E1 -4455.451,E2 -4455.451} C_VEL
LIN {X 0,Y 530.982,Z 178.342,A -85,B 0,C 180,E1 -4458.563,E2 -4458.563} C_VEL
LIN {X 0,Y 530.956,Z 178.343,A -85,B 0,C 180,E1 -4461.529,E2 -4461.529} C_VEL
LIN {X 0,Y 530.956,Z 178.345,A -85,B 0,C 180,E1 -4464.38,E2 -4464.38} C_VEL
LIN {X 0,Y 530.968,Z 178.345,A -85,B 0,C 180,E1 -4467.133,E2 -4467.133} C_VEL
LIN {X 0,Y 530.961,Z 178.342,A -85,B 0,C 180,E1 -4469.802,E2 -4469.802} C_VEL
LIN {X 0,Y 531.011,Z 178.342,A -85,B 0,C 180,E1 -4472.468,E2 -4472.468} C_VEL
LIN {X 0,Y 530.99,Z 178.343,A -85,B 0,C 180,E1 -4474.941,E2 -4474.941} C_VEL
LIN {X 0,Y 530.973,Z 178.344,A -85,B 0,C 180,E1 -4478.246,E2 -4478.246} C_VEL
LIN {X 0,Y 530.986,Z 178.346,A -85,B 0,C 180,E1 -4480.677,E2 -4480.677} C_VEL
LIN {X 0,Y 530.971,Z 178.343,A -85,B 0,C 180,E1 -4483.07,E2 -4483.07} C_VEL
LIN {X 0,Y 531.02,Z 178.335,A -85,B 0,C 180,E1 -4485.436,E2 -4485.436} C_VEL
LIN {X 0,Y 531.036,Z 178.34,A -85,B 0,C 180,E1 -4488.549,E2 -4488.549} C_VEL
LIN {X 0,Y 531.038,Z 178.334,A -85,B 0,C 180,E1 -4491.629,E2 -4491.629} C_VEL
LIN {X 0,Y 531.114,Z 178.328,A -85,B 0,C 180,E1 -4494.685,E2 -4494.685} C_VEL
LIN {X 0,Y 531.136,Z 178.324,A -85,B 0,C 180,E1 -4497.725,E2 -4497.725} C_VEL
LIN {X 0,Y 531.062,Z 178.416,A -85,B 0,C 180,E1 -4500.308,E2 -4500.308} C_VEL
LIN {X 0,Y 531.046,Z 195.962,A -85,B 0,C 180,E1 -4503.224,E2 -4503.224} C_VEL
LIN {X 0,Y 531.01,Z 210.476,A -85,B 0,C 180,E1 -4505.696,E2 -4505.696} C_VEL
LIN {X 0,Y 531.022,Z 224.647,A -85,B 0,C 180,E1 -4508.179,E2 -4508.179} C_VEL
LIN {X 0,Y 532.03,Z 231.274,A -85,B 0,C 180,E1 -4508.331,E2 -4508.331} C_VEL
LIN {X 0,Y 531.804,Z 302.843,A -85,B 0,C 180,E1 -4509.364,E2 -4509.364} C_VEL
LIN {X 0,Y 531.665,Z 315.296,A -85,B 0,C 180,E1 -4509.703,E2 -4509.703} C_VEL
LIN {X 0,Y 531.535,Z 326.693,A -85,B 0,C 180,E1 -4510.186,E2 -4510.186} C_VEL
LIN {X 0,Y 531.393,Z 336.74,A -85,B 0,C 180,E1 -4510.766,E2 -4510.766} C_VEL
LIN {X 0,Y 531.181,Z 347.198,A -85,B 0,C 180,E1 -4511.558,E2 -4511.558} C_VEL
LIN {X 0,Y 531.031,Z 355.985,A -85,B 0,C 180,E1 -4512.419,E2 -4512.419} C_VEL
LIN {X 0,Y 530.854,Z 363.853,A -85,B 0,C 180,E1 -4513.396,E2 -4513.396} C_VEL
LIN {X 0,Y 530.746,Z 370.082,A -85,B 0,C 180,E1 -4514.376,E2 -4514.376} C_VEL
LIN {X 0,Y 530.649,Z 375.009,A -85,B 0,C 180,E1 -4515.36,E2 -4515.36} C_VEL
LIN {X 0,Y 530.587,Z 379.433,A -85,B 0,C 180,E1 -4516.545,E2 -4516.545} C_VEL
LIN {X 0,Y 530.487,Z 382.481,A -85,B 0,C 180,E1 -4517.74,E2 -4517.74} C_VEL
LIN {X 0,Y 530.45,Z 383.779,A -85,B 0,C 180,E1 -4518.54,E2 -4518.54} C_VEL
LIN {X 0,Y 530.479,Z 384.718,A -85,B 0,C 180,E1 -4519.841,E2 -4519.841} C_VEL
LIN {X 0,Y 530.45,Z 384.375,A -85,B 0,C 180,E1 -4520.96,E2 -4520.96} C_VEL
LIN {X 0,Y 530.476,Z 383.133,A -85,B 0,C 180,E1 -4521.968,E2 -4521.968} C_VEL
LIN {X 0,Y 530.504,Z 380.904,A -85,B 0,C 180,E1 -4523.004,E2 -4523.004} C_VEL
LIN {X 0,Y 530.62,Z 376.859,A -85,B 0,C 180,E1 -4524.242,E2 -4524.242} C_VEL
LIN {X 0,Y 530.712,Z 371.466,A -85,B 0,C 180,E1 -4525.427,E2 -4525.427} C_VEL
LIN {X 0,Y 530.806,Z 364.712,A -85,B 0,C 180,E1 -4526.542,E2 -4526.542} C_VEL
LIN {X 0,Y 530.934,Z 357.105,A -85,B 0,C 180,E1 -4527.516,E2 -4527.516} C_VEL
LIN {X 0,Y 531.101,Z 349.026,A -85,B 0,C 180,E1 -4528.341,E2 -4528.341} C_VEL
LIN {X 0,Y 531.306,Z 339.851,A -85,B 0,C 180,E1 -4529.085,E2 -4529.085} C_VEL
LIN {X 0,Y 531.421,Z 333.706,A -85,B 0,C 180,E1 -4529.491,E2 -4529.491} C_VEL
LIN {X 0,Y 530.814,Z 330.302,A -85,B 0,C 180,E1 -4529.708,E2 -4529.708} C_VEL
LIN {X 0,Y 528.052,Z 324.971,A -85,B 0,C 180,E1 -4530.049,E2 -4530.049} C_VEL
LIN {X 0,Y 525.314,Z 319.466,A -85,B 0,C 180,E1 -4530.354,E2 -4530.354} C_VEL
LIN {X 0,Y 524.704,Z 315.795,A -85,B 0,C 180,E1 -4530.507,E2 -4530.507} C_VEL
LIN {X 0,Y 524.772,Z 304.318,A -85,B 0,C 180,E1 -4530.835,E2 -4530.835} C_VEL
LIN {X 0,Y 524.963,Z 267.97,A -85,B 0,C 180,E1 -4531.377,E2 -4531.377} C_VEL
LIN {X 0,Y 524.987,Z 231.101,A -85,B 0,C 180,E1 -4531.904,E2 -4531.904} C_VEL
LIN {X 0,Y 524.012,Z 224.813,A -85,B 0,C 180,E1 -4532.046,E2 -4532.046} C_VEL
LIN {X 0,Y 523.962,Z 221.205,A -85,B 0,C 180,E1 -4532.675,E2 -4532.675} C_VEL
LIN {X 0,Y 524.189,Z 204.159,A -85,B 0,C 180,E1 -4535.914,E2 -4535.914} C_VEL
LIN {X 0,Y 524.368,Z 187.68,A -85,B 0,C 180,E1 -4539.045,E2 -4539.045} C_VEL
LIN {X 0,Y 524.276,Z 180.931,A -85,B 0,C 180,E1 -4540.351,E2 -4540.351} C_VEL
LIN {X 0,Y 524.011,Z 179.237,A -85,B 0,C 180,E1 -4540.759,E2 -4540.759} C_VEL
LIN {X 0,Y 523.917,Z 179.225,A -85,B 0,C 180,E1 -4543.583,E2 -4543.583} C_VEL
LIN {X 0,Y 523.917,Z 179.221,A -85,B 0,C 180,E1 -4546.416,E2 -4546.416} C_VEL
LIN {X 0,Y 523.939,Z 179.216,A -85,B 0,C 180,E1 -4548.907,E2 -4548.907} C_VEL
LIN {X 0,Y 523.914,Z 179.225,A -85,B 0,C 180,E1 -4551.898,E2 -4551.898} C_VEL
LIN {X 0,Y 523.933,Z 179.217,A -85,B 0,C 180,E1 -4554.909,E2 -4554.909} C_VEL
LIN {X 0,Y 523.934,Z 179.224,A -85,B 0,C 180,E1 -4557.679,E2 -4557.679} C_VEL
LIN {X 0,Y 523.952,Z 179.214,A -85,B 0,C 180,E1 -4560.676,E2 -4560.676} C_VEL
LIN {X 0,Y 523.976,Z 179.217,A -85,B 0,C 180,E1 -4563.728,E2 -4563.728} C_VEL
LIN {X 0,Y 523.925,Z 179.218,A -85,B 0,C 180,E1 -4566.27,E2 -4566.27} C_VEL
LIN {X 0,Y 523.944,Z 179.216,A -85,B 0,C 180,E1 -4568.766,E2 -4568.766} C_VEL
LIN {X 0,Y 523.948,Z 179.221,A -85,B 0,C 180,E1 -4571.22,E2 -4571.22} C_VEL
LIN {X 0,Y 523.936,Z 179.221,A -85,B 0,C 180,E1 -4573.638,E2 -4573.638} C_VEL
LIN {X 0,Y 523.943,Z 179.216,A -85,B 0,C 180,E1 -4576.028,E2 -4576.028} C_VEL
LIN {X 0,Y 524.011,Z 179.207,A -85,B 0,C 180,E1 -4578.394,E2 -4578.394} C_VEL
LIN {X 0,Y 524.003,Z 179.212,A -85,B 0,C 180,E1 -4581.516,E2 -4581.516} C_VEL
LIN {X 0,Y 524.084,Z 179.199,A -85,B 0,C 180,E1 -4584.613,E2 -4584.613} C_VEL
LIN {X 0,Y 524.112,Z 179.196,A -85,B 0,C 180,E1 -4587.694,E2 -4587.694} C_VEL
LIN {X 0,Y 524.12,Z 179.198,A -85,B 0,C 180,E1 -4590.768,E2 -4590.768} C_VEL
LIN {X 0,Y 524.069,Z 179.208,A -85,B 0,C 180,E1 -4593.074,E2 -4593.074} C_VEL
LIN {X 0,Y 524.035,Z 179.204,A -85,B 0,C 180,E1 -4596.159,E2 -4596.159} C_VEL
LIN {X 0,Y 524.001,Z 179.211,A -85,B 0,C 180,E1 -4598.483,E2 -4598.483} C_VEL
LIN {X 0,Y 523.999,Z 179.208,A -85,B 0,C 180,E1 -4601.739,E2 -4601.739} C_VEL
LIN {X 0,Y 523.989,Z 179.215,A -85,B 0,C 180,E1 -4605.052,E2 -4605.052} C_VEL
LIN {X 0,Y 523.96,Z 179.213,A -85,B 0,C 180,E1 -4607.968,E2 -4607.968} C_VEL
LIN {X 0,Y 523.967,Z 179.216,A -85,B 0,C 180,E1 -4610.409,E2 -4610.409} C_VEL
LIN {X 0,Y 523.912,Z 179.226,A -85,B 0,C 180,E1 -4612.893,E2 -4612.893} C_VEL
LIN {X 0,Y 523.95,Z 179.215,A -85,B 0,C 180,E1 -4615.418,E2 -4615.418} C_VEL
LIN {X 0,Y 523.966,Z 179.213,A -85,B 0,C 180,E1 -4617.998,E2 -4617.998} C_VEL
LIN {X 0,Y 523.941,Z 179.221,A -85,B 0,C 180,E1 -4620.855,E2 -4620.855} C_VEL
LIN {X 0,Y 523.957,Z 179.214,A -85,B 0,C 180,E1 -4623.735,E2 -4623.735} C_VEL
LIN {X 0,Y 523.918,Z 179.226,A -85,B 0,C 180,E1 -4626.404,E2 -4626.404} C_VEL
LIN {X 0,Y 523.924,Z 179.219,A -85,B 0,C 180,E1 -4629.083,E2 -4629.083} C_VEL
LIN {X 0,Y 523.965,Z 179.212,A -85,B 0,C 180,E1 -4631.312,E2 -4631.312} C_VEL
LIN {X 0,Y 523.948,Z 179.219,A -85,B 0,C 180,E1 -4634.691,E2 -4634.691} C_VEL
LIN {X 0,Y 523.949,Z 179.217,A -85,B 0,C 180,E1 -4637.881,E2 -4637.881} C_VEL
LIN {X 0,Y 523.97,Z 179.215,A -85,B 0,C 180,E1 -4639.923,E2 -4639.923} C_VEL
LIN {X 0,Y 523.903,Z 179.221,A -85,B 0,C 180,E1 -4642.868,E2 -4642.868} C_VEL
LIN {X 0,Y 523.938,Z 179.218,A -85,B 0,C 180,E1 -4645.711,E2 -4645.711} C_VEL
LIN {X 0,Y 523.925,Z 179.222,A -85,B 0,C 180,E1 -4648.457,E2 -4648.457} C_VEL
LIN {X 0,Y 523.942,Z 179.215,A -85,B 0,C 180,E1 -4651.126,E2 -4651.126} C_VEL
LIN {X 0,Y 523.975,Z 179.219,A -85,B 0,C 180,E1 -4653.98,E2 -4653.98} C_VEL
LIN {X 0,Y 523.928,Z 179.223,A -85,B 0,C 180,E1 -4656.271,E2 -4656.271} C_VEL
LIN {X 0,Y 523.939,Z 179.216,A -85,B 0,C 180,E1 -4658.767,E2 -4658.767} C_VEL
LIN {X 0,Y 523.945,Z 179.215,A -85,B 0,C 180,E1 -4661.221,E2 -4661.221} C_VEL
LIN {X 0,Y 523.931,Z 179.221,A -85,B 0,C 180,E1 -4663.639,E2 -4663.639} C_VEL
LIN {X 0,Y 523.932,Z 179.224,A -85,B 0,C 180,E1 -4666.028,E2 -4666.028} C_VEL
LIN {X 0,Y 524.003,Z 179.21,A -85,B 0,C 180,E1 -4668.394,E2 -4668.394} C_VEL
LIN {X 0,Y 523.996,Z 179.213,A -85,B 0,C 180,E1 -4671.516,E2 -4671.516} C_VEL
LIN {X 0,Y 524.074,Z 179.199,A -85,B 0,C 180,E1 -4674.614,E2 -4674.614} C_VEL
LIN {X 0,Y 524.102,Z 179.205,A -85,B 0,C 180,E1 -4677.695,E2 -4677.695} C_VEL
LIN {X 0,Y 524.115,Z 179.194,A -85,B 0,C 180,E1 -4680.769,E2 -4680.769} C_VEL
LIN {X 0,Y 524.065,Z 179.202,A -85,B 0,C 180,E1 -4683.075,E2 -4683.075} C_VEL
LIN {X 0,Y 524.029,Z 179.206,A -85,B 0,C 180,E1 -4686.16,E2 -4686.16} C_VEL
LIN {X 0,Y 523.991,Z 179.209,A -85,B 0,C 180,E1 -4688.485,E2 -4688.485} C_VEL
LIN {X 0,Y 523.994,Z 179.214,A -85,B 0,C 180,E1 -4691.74,E2 -4691.74} C_VEL
LIN {X 0,Y 523.985,Z 179.213,A -85,B 0,C 180,E1 -4695.053,E2 -4695.053} C_VEL
LIN {X 0,Y 523.956,Z 179.215,A -85,B 0,C 180,E1 -4697.97,E2 -4697.97} C_VEL
LIN {X 0,Y 523.964,Z 179.212,A -85,B 0,C 180,E1 -4700.411,E2 -4700.411} C_VEL
LIN {X 0,Y 523.904,Z 179.223,A -85,B 0,C 180,E1 -4702.894,E2 -4702.894} C_VEL
LIN {X 0,Y 523.977,Z 179.211,A -85,B 0,C 180,E1 -4706.02,E2 -4706.02} C_VEL
LIN {X 0,Y 523.923,Z 179.222,A -85,B 0,C 180,E1 -4708.876,E2 -4708.876} C_VEL
LIN {X 0,Y 523.915,Z 179.223,A -85,B 0,C 180,E1 -4711.545,E2 -4711.545} C_VEL
LIN {X 0,Y 523.914,Z 179.219,A -85,B 0,C 180,E1 -4714.292,E2 -4714.292} C_VEL
LIN {X 0,Y 523.901,Z 179.229,A -85,B 0,C 180,E1 -4717.133,E2 -4717.133} C_VEL
LIN {X 0,Y 523.933,Z 179.216,A -85,B 0,C 180,E1 -4720.131,E2 -4720.131} C_VEL
LIN {X 0,Y 523.93,Z 179.219,A -85,B 0,C 180,E1 -4722.46,E2 -4722.46} C_VEL
LIN {X 0,Y 523.948,Z 179.219,A -85,B 0,C 180,E1 -4725.31,E2 -4725.31} C_VEL
LIN {X 0,Y 523.936,Z 179.222,A -85,B 0,C 180,E1 -4728.693,E2 -4728.693} C_VEL
LIN {X 0,Y 523.914,Z 179.225,A -85,B 0,C 180,E1 -4731.082,E2 -4731.082} C_VEL
LIN {X 0,Y 523.892,Z 179.221,A -85,B 0,C 180,E1 -4733.826,E2 -4733.826} C_VEL
LIN {X 0,Y 523.939,Z 179.224,A -85,B 0,C 180,E1 -4736.636,E2 -4736.636} C_VEL
LIN {X 0,Y 523.942,Z 179.219,A -85,B 0,C 180,E1 -4739.356,E2 -4739.356} C_VEL
LIN {X 0,Y 523.945,Z 179.221,A -85,B 0,C 180,E1 -4742.289,E2 -4742.289} C_VEL
LIN {X 0,Y 523.97,Z 179.399,A -85,B 0,C 180,E1 -4744.275,E2 -4744.275} C_VEL
LIN {X 0,Y 526.308,Z 190.377,A -85,B 0,C 180,E1 -4745.757,E2 -4745.757} C_VEL
LIN {X 0,Y 525.675,Z 214.213,A -85,B 0,C 180,E1 -4748.635,E2 -4748.635} C_VEL
LIN {X 0,Y 525.006,Z 241.623,A -85,B 0,C 180,E1 -4751.887,E2 -4751.887} C_VEL
LIN {X 0,Y 524.556,Z 267.53,A -85,B 0,C 180,E1 -4754.903,E2 -4754.903} C_VEL
LIN {X 0,Y 525.713,Z 279.991,A -85,B 0,C 180,E1 -4755.132,E2 -4755.132} C_VEL
LIN {X 0,Y 525.307,Z 376.961,A -85,B 0,C 180,E1 -4756.485,E2 -4756.485} C_VEL
LIN {X 0,Y 525.099,Z 390.296,A -85,B 0,C 180,E1 -4756.824,E2 -4756.824} C_VEL
LIN {X 0,Y 524.881,Z 402.513,A -85,B 0,C 180,E1 -4757.286,E2 -4757.286} C_VEL
LIN {X 0,Y 524.634,Z 414.074,A -85,B 0,C 180,E1 -4757.873,E2 -4757.873} C_VEL
LIN {X 0,Y 524.388,Z 425.176,A -85,B 0,C 180,E1 -4758.599,E2 -4758.599} C_VEL
LIN {X 0,Y 524.118,Z 435.897,A -85,B 0,C 180,E1 -4759.474,E2 -4759.474} C_VEL
LIN {X 0,Y 523.901,Z 444.654,A -85,B 0,C 180,E1 -4760.347,E2 -4760.347} C_VEL
LIN {X 0,Y 523.737,Z 452.722,A -85,B 0,C 180,E1 -4761.318,E2 -4761.318} C_VEL
LIN {X 0,Y 523.577,Z 460.609,A -85,B 0,C 180,E1 -4762.48,E2 -4762.48} C_VEL
LIN {X 0,Y 523.467,Z 467.842,A -85,B 0,C 180,E1 -4763.835,E2 -4763.835} C_VEL
LIN {X 0,Y 523.383,Z 472.656,A -85,B 0,C 180,E1 -4764.993,E2 -4764.993} C_VEL
LIN {X 0,Y 523.443,Z 476.344,A -85,B 0,C 180,E1 -4766.151,E2 -4766.151} C_VEL
LIN {X 0,Y 523.446,Z 478.242,A -85,B 0,C 180,E1 -4766.922,E2 -4766.922} C_VEL
LIN {X 0,Y 523.344,Z 479.656,A -85,B 0,C 180,E1 -4767.692,E2 -4767.692} C_VEL
LIN {X 0,Y 523.301,Z 481.279,A -85,B 0,C 180,E1 -4769.231,E2 -4769.231} C_VEL
LIN {X 0,Y 523.305,Z 481.494,A -85,B 0,C 180,E1 -4770.001,E2 -4770.001} C_VEL
LIN {X 0,Y 523.302,Z 481.267,A -85,B 0,C 180,E1 -4770.77,E2 -4770.77} C_VEL
LIN {X 0,Y 523.346,Z 479.624,A -85,B 0,C 180,E1 -4772.309,E2 -4772.309} C_VEL
LIN {X 0,Y 523.446,Z 478.195,A -85,B 0,C 180,E1 -4773.079,E2 -4773.079} C_VEL
LIN {X 0,Y 523.443,Z 475.184,A -85,B 0,C 180,E1 -4774.235,E2 -4774.235} C_VEL
LIN {X 0,Y 523.464,Z 471.11,A -85,B 0,C 180,E1 -4775.393,E2 -4775.393} C_VEL
LIN {X 0,Y 523.538,Z 464.873,A -85,B 0,C 180,E1 -4776.739,E2 -4776.739} C_VEL
LIN {X 0,Y 523.657,Z 457.992,A -85,B 0,C 180,E1 -4777.907,E2 -4777.907} C_VEL
LIN {X 0,Y 523.795,Z 449.481,A -85,B 0,C 180,E1 -4779.071,E2 -4779.071} C_VEL
LIN {X 0,Y 523.972,Z 440.711,A -85,B 0,C 180,E1 -4780.042,E2 -4780.042} C_VEL
LIN {X 0,Y 524.225,Z 429.903,A -85,B 0,C 180,E1 -4781.014,E2 -4781.014} C_VEL
LIN {X 0,Y 524.499,Z 418.347,A -85,B 0,C 180,E1 -4781.844,E2 -4781.844} C_VEL
LIN {X 0,Y 524.726,Z 406.154,A -85,B 0,C 180,E1 -4782.522,E2 -4782.522} C_VEL
LIN {X 0,Y 525.02,Z 393.345,A -85,B 0,C 180,E1 -4783.056,E2 -4783.056} C_VEL
LIN {X 0,Y 525.233,Z 380.657,A -85,B 0,C 180,E1 -4783.42,E2 -4783.42} C_VEL
LIN {X 0,Y 525.354,Z 362.7,A -85,B 0,C 180,E1 -4783.712,E2 -4783.712} C_VEL
LIN {X 0,Y 525.575,Z 276.938,A -85,B 0,C 180,E1 -4784.901,E2 -4784.901} C_VEL
LIN {X 0,Y 524.494,Z 267.154,A -85,B 0,C 180,E1 -4785.089,E2 -4785.089} C_VEL
LIN {X 0,Y 524.928,Z 240.836,A -85,B 0,C 180,E1 -4788.087,E2 -4788.087} C_VEL
LIN {X 0,Y 525.442,Z 212.37,A -85,B 0,C 180,E1 -4791.376,E2 -4791.376} C_VEL
LIN {X 0,Y 525.871,Z 189.341,A -85,B 0,C 180,E1 -4794.056,E2 -4794.056} C_VEL
LIN {X 0,Y 523.973,Z 179.353,A -85,B 0,C 180,E1 -4795.351,E2 -4795.351} C_VEL
LIN {X 0,Y 523.914,Z 179.224,A -85,B 0,C 180,E1 -4798.002,E2 -4798.002} C_VEL
LIN {X 0,Y 523.938,Z 179.223,A -85,B 0,C 180,E1 -4800.853,E2 -4800.853} C_VEL
LIN {X 0,Y 523.932,Z 179.221,A -85,B 0,C 180,E1 -4803.729,E2 -4803.729} C_VEL
LIN {X 0,Y 523.901,Z 179.223,A -85,B 0,C 180,E1 -4806.4,E2 -4806.4} C_VEL
LIN {X 0,Y 523.915,Z 179.228,A -85,B 0,C 180,E1 -4809.085,E2 -4809.085} C_VEL
LIN {X 0,Y 523.914,Z 179.22,A -85,B 0,C 180,E1 -4812.123,E2 -4812.123} C_VEL
